(* Logix 5000 project; controller reports 1756-L63 rev 20.11; software revision 20.04; part 9 of 52 *)

        [41].log_data[16].valid := 1, [41].log_data[17].valid := 1, [41].log_data[18].valid := 1, [41].log_data[19].valid := 1, [41].time.Year := 2023, [41].time.Month := 1, [41].time.Day := 18, [41].time.Hour := 3, [41].time.Minute := 49, [41].time.Second := 59, [42].log_data[0].min := 1.0, [42].log_data[0].max := 1.0, [42].log_data[0].total := 300.0, [42].log_data[0].time := 300.0, [42].log_data[0].minminute := 50, [42].log_data[0].maxminute := 50, [42].log_data[0].valid := 1, [42].log_data[1].valid := 1, [42].log_data[2].valid := 1, [42].log_data[3].valid := 1, [42].log_data[4].valid := 1, [42].log_data[5].valid := 1, [42].log_data[6].valid := 1, [42].log_data[7].valid := 1, [42].log_data[8].valid := 1, [42].log_data[9].valid := 1, [42].log_data[10].valid := 1, [42].log_data[11].valid := 1, [42].log_data[12].valid := 1, [42].log_data[13].valid := 1, [42].log_data[14].valid := 1, [42].log_data[15].valid := 1, [42].log_data[16].valid := 1, [42].log_data[17].valid := 1, [42].log_data[18].valid := 1, [42].log_data[19].valid := 1, [42].time.Year := 2023, [42].time.Month := 1, [42].time.Day := 18, [42].time.Hour := 3, [42].time.Minute := 54, [42].time.Second := 59, [43].log_data[0].min := 1.0, [43].log_data[0].max := 1.0, [43].log_data[0].total := 300.0, [43].log_data[0].time := 300.0, [43].log_data[0].minminute := 55, [43].log_data[0].maxminute := 55, [43].log_data[0].valid := 1, [43].log_data[1].valid := 1, [43].log_data[2].valid := 1, [43].log_data[3].valid := 1, [43].log_data[4].valid := 1, [43].log_data[5].valid := 1, [43].log_data[6].valid := 1, [43].log_data[7].valid := 1, [43].log_data[8].valid := 1, [43].log_data[9].valid := 1, [43].log_data[10].valid := 1, [43].log_data[11].valid := 1,
        [43].log_data[12].valid := 1, [43].log_data[13].valid := 1, [43].log_data[14].valid := 1, [43].log_data[15].valid := 1, [43].log_data[16].valid := 1, [43].log_data[17].valid := 1, [43].log_data[18].valid := 1, [43].log_data[19].valid := 1, [43].time.Year := 2023, [43].time.Month := 1, [43].time.Day := 18, [43].time.Hour := 3, [43].time.Minute := 59, [43].time.Second := 59, [44].log_data[0].min := 1.0, [44].log_data[0].max := 1.0, [44].log_data[0].total := 300.0, [44].log_data[0].time := 300.0, [44].log_data[0].valid := 1, [44].log_data[1].valid := 1, [44].log_data[2].valid := 1, [44].log_data[3].valid := 1, [44].log_data[4].valid := 1, [44].log_data[5].valid := 1, [44].log_data[6].valid := 1, [44].log_data[7].valid := 1, [44].log_data[8].valid := 1, [44].log_data[9].valid := 1, [44].log_data[10].valid := 1, [44].log_data[11].valid := 1, [44].log_data[12].valid := 1, [44].log_data[13].valid := 1, [44].log_data[14].valid := 1, [44].log_data[15].valid := 1, [44].log_data[16].valid := 1, [44].log_data[17].valid := 1, [44].log_data[18].valid := 1, [44].log_data[19].valid := 1, [44].time.Year := 2023, [44].time.Month := 1, [44].time.Day := 18, [44].time.Hour := 4, [44].time.Minute := 4, [44].time.Second := 59, [45].log_data[0].min := 1.0, [45].log_data[0].max := 1.0, [45].log_data[0].total := 300.0, [45].log_data[0].time := 300.0, [45].log_data[0].minminute := 5, [45].log_data[0].maxminute := 5, [45].log_data[0].valid := 1, [45].log_data[1].valid := 1, [45].log_data[2].valid := 1, [45].log_data[3].valid := 1, [45].log_data[4].valid := 1, [45].log_data[5].valid := 1, [45].log_data[6].valid := 1, [45].log_data[7].valid := 1, [45].log_data[8].valid := 1, [45].log_data[9].valid := 1,
        [45].log_data[10].valid := 1, [45].log_data[11].valid := 1, [45].log_data[12].valid := 1, [45].log_data[13].valid := 1, [45].log_data[14].valid := 1, [45].log_data[15].valid := 1, [45].log_data[16].valid := 1, [45].log_data[17].valid := 1, [45].log_data[18].valid := 1, [45].log_data[19].valid := 1, [45].time.Year := 2023, [45].time.Month := 1, [45].time.Day := 18, [45].time.Hour := 4, [45].time.Minute := 9, [45].time.Second := 59, [46].log_data[0].min := 1.0, [46].log_data[0].max := 1.0, [46].log_data[0].total := 300.0, [46].log_data[0].time := 300.0, [46].log_data[0].minminute := 10, [46].log_data[0].maxminute := 10, [46].log_data[0].valid := 1, [46].log_data[1].valid := 1, [46].log_data[2].valid := 1, [46].log_data[3].valid := 1, [46].log_data[4].valid := 1, [46].log_data[5].valid := 1, [46].log_data[6].valid := 1, [46].log_data[7].valid := 1, [46].log_data[8].valid := 1, [46].log_data[9].valid := 1, [46].log_data[10].valid := 1, [46].log_data[11].valid := 1, [46].log_data[12].valid := 1, [46].log_data[13].valid := 1, [46].log_data[14].valid := 1, [46].log_data[15].valid := 1, [46].log_data[16].valid := 1, [46].log_data[17].valid := 1, [46].log_data[18].valid := 1, [46].log_data[19].valid := 1, [46].time.Year := 2023, [46].time.Month := 1, [46].time.Day := 18, [46].time.Hour := 4, [46].time.Minute := 14, [46].time.Second := 59, [47].log_data[0].min := 1.0, [47].log_data[0].max := 1.0, [47].log_data[0].total := 300.0, [47].log_data[0].time := 300.0, [47].log_data[0].minminute := 15, [47].log_data[0].maxminute := 15, [47].log_data[0].valid := 1, [47].log_data[1].valid := 1, [47].log_data[2].valid := 1, [47].log_data[3].valid := 1, [47].log_data[4].valid := 1, [47].log_data[5].valid := 1,
        [47].log_data[6].valid := 1, [47].log_data[7].valid := 1, [47].log_data[8].valid := 1, [47].log_data[9].valid := 1, [47].log_data[10].valid := 1, [47].log_data[11].valid := 1, [47].log_data[12].valid := 1, [47].log_data[13].valid := 1, [47].log_data[14].valid := 1, [47].log_data[15].valid := 1, [47].log_data[16].valid := 1, [47].log_data[17].valid := 1, [47].log_data[18].valid := 1, [47].log_data[19].valid := 1, [47].time.Year := 2023, [47].time.Month := 1, [47].time.Day := 18, [47].time.Hour := 4, [47].time.Minute := 19, [47].time.Second := 59, [48].log_data[0].min := 1.0, [48].log_data[0].max := 1.0, [48].log_data[0].total := 300.0, [48].log_data[0].time := 300.0, [48].log_data[0].minminute := 20, [48].log_data[0].maxminute := 20, [48].log_data[0].valid := 1, [48].log_data[1].valid := 1, [48].log_data[2].valid := 1, [48].log_data[3].valid := 1, [48].log_data[4].valid := 1, [48].log_data[5].valid := 1, [48].log_data[6].valid := 1, [48].log_data[7].valid := 1, [48].log_data[8].valid := 1, [48].log_data[9].valid := 1, [48].log_data[10].valid := 1, [48].log_data[11].valid := 1, [48].log_data[12].valid := 1, [48].log_data[13].valid := 1, [48].log_data[14].valid := 1, [48].log_data[15].valid := 1, [48].log_data[16].valid := 1, [48].log_data[17].valid := 1, [48].log_data[18].valid := 1, [48].log_data[19].valid := 1, [48].time.Year := 2023, [48].time.Month := 1, [48].time.Day := 18, [48].time.Hour := 4, [48].time.Minute := 24, [48].time.Second := 59, [49].log_data[0].min := 1.0, [49].log_data[0].max := 1.0, [49].log_data[0].total := 300.0, [49].log_data[0].time := 300.0, [49].log_data[0].minminute := 25, [49].log_data[0].maxminute := 25, [49].log_data[0].valid := 1, [49].log_data[1].valid := 1,
        [49].log_data[2].valid := 1, [49].log_data[3].valid := 1, [49].log_data[4].valid := 1, [49].log_data[5].valid := 1, [49].log_data[6].valid := 1, [49].log_data[7].valid := 1, [49].log_data[8].valid := 1, [49].log_data[9].valid := 1, [49].log_data[10].valid := 1, [49].log_data[11].valid := 1, [49].log_data[12].valid := 1, [49].log_data[13].valid := 1, [49].log_data[14].valid := 1, [49].log_data[15].valid := 1, [49].log_data[16].valid := 1, [49].log_data[17].valid := 1, [49].log_data[18].valid := 1, [49].log_data[19].valid := 1, [49].time.Year := 2023, [49].time.Month := 1, [49].time.Day := 18, [49].time.Hour := 4, [49].time.Minute := 29, [49].time.Second := 59, [50].log_data[0].min := 1.0, [50].log_data[0].max := 1.0, [50].log_data[0].total := 300.0, [50].log_data[0].time := 300.0, [50].log_data[0].minminute := 30, [50].log_data[0].maxminute := 30, [50].log_data[0].valid := 1, [50].log_data[1].valid := 1, [50].log_data[2].valid := 1, [50].log_data[3].valid := 1, [50].log_data[4].valid := 1, [50].log_data[5].valid := 1, [50].log_data[6].valid := 1, [50].log_data[7].valid := 1, [50].log_data[8].valid := 1, [50].log_data[9].valid := 1, [50].log_data[10].valid := 1, [50].log_data[11].valid := 1, [50].log_data[12].valid := 1, [50].log_data[13].valid := 1, [50].log_data[14].valid := 1, [50].log_data[15].valid := 1, [50].log_data[16].valid := 1, [50].log_data[17].valid := 1, [50].log_data[18].valid := 1, [50].log_data[19].valid := 1, [50].time.Year := 2023, [50].time.Month := 1, [50].time.Day := 18, [50].time.Hour := 4, [50].time.Minute := 34, [50].time.Second := 59, [51].log_data[0].min := 1.0, [51].log_data[0].max := 1.0, [51].log_data[0].total := 300.0, [51].log_data[0].time := 300.0,
        [51].log_data[0].minminute := 35, [51].log_data[0].maxminute := 35, [51].log_data[0].valid := 1, [51].log_data[1].valid := 1, [51].log_data[2].valid := 1, [51].log_data[3].valid := 1, [51].log_data[4].valid := 1, [51].log_data[5].valid := 1, [51].log_data[6].valid := 1, [51].log_data[7].valid := 1, [51].log_data[8].valid := 1, [51].log_data[9].valid := 1, [51].log_data[10].valid := 1, [51].log_data[11].valid := 1, [51].log_data[12].valid := 1, [51].log_data[13].valid := 1, [51].log_data[14].valid := 1, [51].log_data[15].valid := 1, [51].log_data[16].valid := 1, [51].log_data[17].valid := 1, [51].log_data[18].valid := 1, [51].log_data[19].valid := 1, [51].time.Year := 2023, [51].time.Month := 1, [51].time.Day := 18, [51].time.Hour := 4, [51].time.Minute := 39, [51].time.Second := 59, [52].log_data[0].min := 1.0, [52].log_data[0].max := 1.0, [52].log_data[0].total := 300.0, [52].log_data[0].time := 300.0, [52].log_data[0].minminute := 40, [52].log_data[0].maxminute := 40, [52].log_data[0].valid := 1, [52].log_data[1].valid := 1, [52].log_data[2].valid := 1, [52].log_data[3].valid := 1, [52].log_data[4].valid := 1, [52].log_data[5].valid := 1, [52].log_data[6].valid := 1, [52].log_data[7].valid := 1, [52].log_data[8].valid := 1, [52].log_data[9].valid := 1, [52].log_data[10].valid := 1, [52].log_data[11].valid := 1, [52].log_data[12].valid := 1, [52].log_data[13].valid := 1, [52].log_data[14].valid := 1, [52].log_data[15].valid := 1, [52].log_data[16].valid := 1, [52].log_data[17].valid := 1, [52].log_data[18].valid := 1, [52].log_data[19].valid := 1, [52].time.Year := 2023, [52].time.Month := 1, [52].time.Day := 18, [52].time.Hour := 4, [52].time.Minute := 44, [52].time.Second := 59,
        [53].log_data[0].min := 1.0, [53].log_data[0].max := 1.0, [53].log_data[0].total := 300.0, [53].log_data[0].time := 300.0, [53].log_data[0].minminute := 45, [53].log_data[0].maxminute := 45, [53].log_data[0].valid := 1, [53].log_data[1].valid := 1, [53].log_data[2].valid := 1, [53].log_data[3].valid := 1, [53].log_data[4].valid := 1, [53].log_data[5].valid := 1, [53].log_data[6].valid := 1, [53].log_data[7].valid := 1, [53].log_data[8].valid := 1, [53].log_data[9].valid := 1, [53].log_data[10].valid := 1, [53].log_data[11].valid := 1, [53].log_data[12].valid := 1, [53].log_data[13].valid := 1, [53].log_data[14].valid := 1, [53].log_data[15].valid := 1, [53].log_data[16].valid := 1, [53].log_data[17].valid := 1, [53].log_data[18].valid := 1, [53].log_data[19].valid := 1, [53].time.Year := 2023, [53].time.Month := 1, [53].time.Day := 18, [53].time.Hour := 4, [53].time.Minute := 49, [53].time.Second := 59, [54].log_data[0].min := 1.0, [54].log_data[0].max := 1.0, [54].log_data[0].total := 300.0, [54].log_data[0].time := 300.0, [54].log_data[0].minminute := 50, [54].log_data[0].maxminute := 50, [54].log_data[0].valid := 1, [54].log_data[1].valid := 1, [54].log_data[2].valid := 1, [54].log_data[3].valid := 1, [54].log_data[4].valid := 1, [54].log_data[5].valid := 1, [54].log_data[6].valid := 1, [54].log_data[7].valid := 1, [54].log_data[8].valid := 1, [54].log_data[9].valid := 1, [54].log_data[10].valid := 1, [54].log_data[11].valid := 1, [54].log_data[12].valid := 1, [54].log_data[13].valid := 1, [54].log_data[14].valid := 1, [54].log_data[15].valid := 1, [54].log_data[16].valid := 1, [54].log_data[17].valid := 1, [54].log_data[18].valid := 1, [54].log_data[19].valid := 1, [54].time.Year := 2023, [54].time.Month := 1,
        [54].time.Day := 18, [54].time.Hour := 4, [54].time.Minute := 54, [54].time.Second := 59, [55].log_data[0].min := 1.0, [55].log_data[0].max := 1.0, [55].log_data[0].total := 300.0, [55].log_data[0].time := 300.0, [55].log_data[0].minminute := 55, [55].log_data[0].maxminute := 55, [55].log_data[0].valid := 1, [55].log_data[1].valid := 1, [55].log_data[2].valid := 1, [55].log_data[3].valid := 1, [55].log_data[4].valid := 1, [55].log_data[5].valid := 1, [55].log_data[6].valid := 1, [55].log_data[7].valid := 1, [55].log_data[8].valid := 1, [55].log_data[9].valid := 1, [55].log_data[10].valid := 1, [55].log_data[11].valid := 1, [55].log_data[12].valid := 1, [55].log_data[13].valid := 1, [55].log_data[14].valid := 1, [55].log_data[15].valid := 1, [55].log_data[16].valid := 1, [55].log_data[17].valid := 1, [55].log_data[18].valid := 1, [55].log_data[19].valid := 1, [55].time.Year := 2023, [55].time.Month := 1, [55].time.Day := 18, [55].time.Hour := 4, [55].time.Minute := 59, [55].time.Second := 59, [56].log_data[0].min := 1.0, [56].log_data[0].max := 1.0, [56].log_data[0].total := 300.0, [56].log_data[0].time := 300.0, [56].log_data[0].valid := 1, [56].log_data[1].valid := 1, [56].log_data[2].valid := 1, [56].log_data[3].valid := 1, [56].log_data[4].valid := 1, [56].log_data[5].valid := 1, [56].log_data[6].valid := 1, [56].log_data[7].valid := 1, [56].log_data[8].valid := 1, [56].log_data[9].valid := 1, [56].log_data[10].valid := 1, [56].log_data[11].valid := 1, [56].log_data[12].valid := 1, [56].log_data[13].valid := 1, [56].log_data[14].valid := 1, [56].log_data[15].valid := 1, [56].log_data[16].valid := 1, [56].log_data[17].valid := 1, [56].log_data[18].valid := 1, [56].log_data[19].valid := 1,
        [56].time.Year := 2023, [56].time.Month := 1, [56].time.Day := 18, [56].time.Hour := 5, [56].time.Minute := 4, [56].time.Second := 59, [57].log_data[0].min := 1.0, [57].log_data[0].max := 1.0, [57].log_data[0].total := 300.0, [57].log_data[0].time := 300.0, [57].log_data[0].minminute := 5, [57].log_data[0].maxminute := 5, [57].log_data[0].valid := 1, [57].log_data[1].valid := 1, [57].log_data[2].valid := 1, [57].log_data[3].valid := 1, [57].log_data[4].valid := 1, [57].log_data[5].valid := 1, [57].log_data[6].valid := 1, [57].log_data[7].valid := 1, [57].log_data[8].valid := 1, [57].log_data[9].valid := 1, [57].log_data[10].valid := 1, [57].log_data[11].valid := 1, [57].log_data[12].valid := 1, [57].log_data[13].valid := 1, [57].log_data[14].valid := 1, [57].log_data[15].valid := 1, [57].log_data[16].valid := 1, [57].log_data[17].valid := 1, [57].log_data[18].valid := 1, [57].log_data[19].valid := 1, [57].time.Year := 2023, [57].time.Month := 1, [57].time.Day := 18, [57].time.Hour := 5, [57].time.Minute := 9, [57].time.Second := 59, [58].log_data[0].min := 1.0, [58].log_data[0].max := 1.0, [58].log_data[0].total := 300.0, [58].log_data[0].time := 300.0, [58].log_data[0].minminute := 10, [58].log_data[0].maxminute := 10, [58].log_data[0].valid := 1, [58].log_data[1].valid := 1, [58].log_data[2].valid := 1, [58].log_data[3].valid := 1, [58].log_data[4].valid := 1, [58].log_data[5].valid := 1, [58].log_data[6].valid := 1, [58].log_data[7].valid := 1, [58].log_data[8].valid := 1, [58].log_data[9].valid := 1, [58].log_data[10].valid := 1, [58].log_data[11].valid := 1, [58].log_data[12].valid := 1, [58].log_data[13].valid := 1, [58].log_data[14].valid := 1, [58].log_data[15].valid := 1,
        [58].log_data[16].valid := 1, [58].log_data[17].valid := 1, [58].log_data[18].valid := 1, [58].log_data[19].valid := 1, [58].time.Year := 2023, [58].time.Month := 1, [58].time.Day := 18, [58].time.Hour := 5, [58].time.Minute := 14, [58].time.Second := 59, [59].log_data[0].min := 1.0, [59].log_data[0].max := 1.0, [59].log_data[0].total := 300.0, [59].log_data[0].time := 300.0, [59].log_data[0].minminute := 15, [59].log_data[0].maxminute := 15, [59].log_data[0].valid := 1, [59].log_data[1].valid := 1, [59].log_data[2].valid := 1, [59].log_data[3].valid := 1, [59].log_data[4].valid := 1, [59].log_data[5].valid := 1, [59].log_data[6].valid := 1, [59].log_data[7].valid := 1, [59].log_data[8].valid := 1, [59].log_data[9].valid := 1, [59].log_data[10].valid := 1, [59].log_data[11].valid := 1, [59].log_data[12].valid := 1, [59].log_data[13].valid := 1, [59].log_data[14].valid := 1, [59].log_data[15].valid := 1, [59].log_data[16].valid := 1, [59].log_data[17].valid := 1, [59].log_data[18].valid := 1, [59].log_data[19].valid := 1, [59].time.Year := 2023, [59].time.Month := 1, [59].time.Day := 18, [59].time.Hour := 5, [59].time.Minute := 19, [59].time.Second := 59, [60].log_data[0].min := 1.0, [60].log_data[0].max := 1.0, [60].log_data[0].total := 300.0, [60].log_data[0].time := 300.0, [60].log_data[0].minminute := 20, [60].log_data[0].maxminute := 20, [60].log_data[0].valid := 1, [60].log_data[1].valid := 1, [60].log_data[2].valid := 1, [60].log_data[3].valid := 1, [60].log_data[4].valid := 1, [60].log_data[5].valid := 1, [60].log_data[6].valid := 1, [60].log_data[7].valid := 1, [60].log_data[8].valid := 1, [60].log_data[9].valid := 1, [60].log_data[10].valid := 1, [60].log_data[11].valid := 1,
        [60].log_data[12].valid := 1, [60].log_data[13].valid := 1, [60].log_data[14].valid := 1, [60].log_data[15].valid := 1, [60].log_data[16].valid := 1, [60].log_data[17].valid := 1, [60].log_data[18].valid := 1, [60].log_data[19].valid := 1, [60].time.Year := 2023, [60].time.Month := 1, [60].time.Day := 18, [60].time.Hour := 5, [60].time.Minute := 24, [60].time.Second := 59, [61].log_data[0].min := 1.0, [61].log_data[0].max := 1.0, [61].log_data[0].total := 300.0, [61].log_data[0].time := 300.0, [61].log_data[0].minminute := 25, [61].log_data[0].maxminute := 25, [61].log_data[0].valid := 1, [61].log_data[1].valid := 1, [61].log_data[2].valid := 1, [61].log_data[3].valid := 1, [61].log_data[4].valid := 1, [61].log_data[5].valid := 1, [61].log_data[6].valid := 1, [61].log_data[7].valid := 1, [61].log_data[8].valid := 1, [61].log_data[9].valid := 1, [61].log_data[10].valid := 1, [61].log_data[11].valid := 1, [61].log_data[12].valid := 1, [61].log_data[13].valid := 1, [61].log_data[14].valid := 1, [61].log_data[15].valid := 1, [61].log_data[16].valid := 1, [61].log_data[17].valid := 1, [61].log_data[18].valid := 1, [61].log_data[19].valid := 1, [61].time.Year := 2023, [61].time.Month := 1, [61].time.Day := 18, [61].time.Hour := 5, [61].time.Minute := 29, [61].time.Second := 59, [62].log_data[0].min := 1.0, [62].log_data[0].max := 1.0, [62].log_data[0].total := 300.0, [62].log_data[0].time := 300.0, [62].log_data[0].minminute := 30, [62].log_data[0].maxminute := 30, [62].log_data[0].valid := 1, [62].log_data[1].valid := 1, [62].log_data[2].valid := 1, [62].log_data[3].valid := 1, [62].log_data[4].valid := 1, [62].log_data[5].valid := 1, [62].log_data[6].valid := 1, [62].log_data[7].valid := 1,
        [62].log_data[8].valid := 1, [62].log_data[9].valid := 1, [62].log_data[10].valid := 1, [62].log_data[11].valid := 1, [62].log_data[12].valid := 1, [62].log_data[13].valid := 1, [62].log_data[14].valid := 1, [62].log_data[15].valid := 1, [62].log_data[16].valid := 1, [62].log_data[17].valid := 1, [62].log_data[18].valid := 1, [62].log_data[19].valid := 1, [62].time.Year := 2023, [62].time.Month := 1, [62].time.Day := 18, [62].time.Hour := 5, [62].time.Minute := 34, [62].time.Second := 59, [63].log_data[0].min := 1.0, [63].log_data[0].max := 1.0, [63].log_data[0].total := 300.0, [63].log_data[0].time := 300.0, [63].log_data[0].minminute := 35, [63].log_data[0].maxminute := 35, [63].log_data[0].valid := 1, [63].log_data[1].valid := 1, [63].log_data[2].valid := 1, [63].log_data[3].valid := 1, [63].log_data[4].valid := 1, [63].log_data[5].valid := 1, [63].log_data[6].valid := 1, [63].log_data[7].valid := 1, [63].log_data[8].valid := 1, [63].log_data[9].valid := 1, [63].log_data[10].valid := 1, [63].log_data[11].valid := 1, [63].log_data[12].valid := 1, [63].log_data[13].valid := 1, [63].log_data[14].valid := 1, [63].log_data[15].valid := 1, [63].log_data[16].valid := 1, [63].log_data[17].valid := 1, [63].log_data[18].valid := 1, [63].log_data[19].valid := 1, [63].time.Year := 2023, [63].time.Month := 1, [63].time.Day := 18, [63].time.Hour := 5, [63].time.Minute := 39, [63].time.Second := 59, [64].log_data[0].min := 1.0, [64].log_data[0].max := 1.0, [64].log_data[0].total := 300.0, [64].log_data[0].time := 300.0, [64].log_data[0].minminute := 40, [64].log_data[0].maxminute := 40, [64].log_data[0].valid := 1, [64].log_data[1].valid := 1, [64].log_data[2].valid := 1, [64].log_data[3].valid := 1,
        [64].log_data[4].valid := 1, [64].log_data[5].valid := 1, [64].log_data[6].valid := 1, [64].log_data[7].valid := 1, [64].log_data[8].valid := 1, [64].log_data[9].valid := 1, [64].log_data[10].valid := 1, [64].log_data[11].valid := 1, [64].log_data[12].valid := 1, [64].log_data[13].valid := 1, [64].log_data[14].valid := 1, [64].log_data[15].valid := 1, [64].log_data[16].valid := 1, [64].log_data[17].valid := 1, [64].log_data[18].valid := 1, [64].log_data[19].valid := 1, [64].time.Year := 2023, [64].time.Month := 1, [64].time.Day := 18, [64].time.Hour := 5, [64].time.Minute := 44, [64].time.Second := 59, [65].log_data[0].min := 1.0, [65].log_data[0].max := 1.0, [65].log_data[0].total := 300.0, [65].log_data[0].time := 300.0, [65].log_data[0].minminute := 45, [65].log_data[0].maxminute := 45, [65].log_data[0].valid := 1, [65].log_data[1].valid := 1, [65].log_data[2].valid := 1, [65].log_data[3].valid := 1, [65].log_data[4].valid := 1, [65].log_data[5].valid := 1, [65].log_data[6].valid := 1, [65].log_data[7].valid := 1, [65].log_data[8].valid := 1, [65].log_data[9].valid := 1, [65].log_data[10].valid := 1, [65].log_data[11].valid := 1, [65].log_data[12].valid := 1, [65].log_data[13].valid := 1, [65].log_data[14].valid := 1, [65].log_data[15].valid := 1, [65].log_data[16].valid := 1, [65].log_data[17].valid := 1, [65].log_data[18].valid := 1, [65].log_data[19].valid := 1, [65].time.Year := 2023, [65].time.Month := 1, [65].time.Day := 18, [65].time.Hour := 5, [65].time.Minute := 49, [65].time.Second := 59, [66].log_data[0].min := 1.0, [66].log_data[0].max := 1.0, [66].log_data[0].total := 300.0, [66].log_data[0].time := 300.0, [66].log_data[0].minminute := 50, [66].log_data[0].maxminute := 50,
        [66].log_data[0].valid := 1, [66].log_data[1].valid := 1, [66].log_data[2].valid := 1, [66].log_data[3].valid := 1, [66].log_data[4].valid := 1, [66].log_data[5].valid := 1, [66].log_data[6].valid := 1, [66].log_data[7].valid := 1, [66].log_data[8].valid := 1, [66].log_data[9].valid := 1, [66].log_data[10].valid := 1, [66].log_data[11].valid := 1, [66].log_data[12].valid := 1, [66].log_data[13].valid := 1, [66].log_data[14].valid := 1, [66].log_data[15].valid := 1, [66].log_data[16].valid := 1, [66].log_data[17].valid := 1, [66].log_data[18].valid := 1, [66].log_data[19].valid := 1, [66].time.Year := 2023, [66].time.Month := 1, [66].time.Day := 18, [66].time.Hour := 5, [66].time.Minute := 54, [66].time.Second := 59, [67].log_data[0].min := 1.0, [67].log_data[0].max := 1.0, [67].log_data[0].total := 300.0, [67].log_data[0].time := 300.0, [67].log_data[0].minminute := 55, [67].log_data[0].maxminute := 55, [67].log_data[0].valid := 1, [67].log_data[1].valid := 1, [67].log_data[2].valid := 1, [67].log_data[3].valid := 1, [67].log_data[4].valid := 1, [67].log_data[5].valid := 1, [67].log_data[6].valid := 1, [67].log_data[7].valid := 1, [67].log_data[8].valid := 1, [67].log_data[9].valid := 1, [67].log_data[10].valid := 1, [67].log_data[11].valid := 1, [67].log_data[12].valid := 1, [67].log_data[13].valid := 1, [67].log_data[14].valid := 1, [67].log_data[15].valid := 1, [67].log_data[16].valid := 1, [67].log_data[17].valid := 1, [67].log_data[18].valid := 1, [67].log_data[19].valid := 1, [67].time.Year := 2023, [67].time.Month := 1, [67].time.Day := 18, [67].time.Hour := 5, [67].time.Minute := 59, [67].time.Second := 59, [68].log_data[0].min := 1.0, [68].log_data[0].max := 1.0,
        [68].log_data[0].total := 300.0, [68].log_data[0].time := 300.0, [68].log_data[0].valid := 1, [68].log_data[1].valid := 1, [68].log_data[2].valid := 1, [68].log_data[3].valid := 1, [68].log_data[4].valid := 1, [68].log_data[5].valid := 1, [68].log_data[6].valid := 1, [68].log_data[7].valid := 1, [68].log_data[8].valid := 1, [68].log_data[9].valid := 1, [68].log_data[10].valid := 1, [68].log_data[11].valid := 1, [68].log_data[12].valid := 1, [68].log_data[13].valid := 1, [68].log_data[14].valid := 1, [68].log_data[15].valid := 1, [68].log_data[16].valid := 1, [68].log_data[17].valid := 1, [68].log_data[18].valid := 1, [68].log_data[19].valid := 1, [68].time.Year := 2023, [68].time.Month := 1, [68].time.Day := 18, [68].time.Hour := 6, [68].time.Minute := 4, [68].time.Second := 59, [69].log_data[0].min := 1.0, [69].log_data[0].max := 1.0, [69].log_data[0].total := 300.0, [69].log_data[0].time := 300.0, [69].log_data[0].minminute := 5, [69].log_data[0].maxminute := 5, [69].log_data[0].valid := 1, [69].log_data[1].valid := 1, [69].log_data[2].valid := 1, [69].log_data[3].valid := 1, [69].log_data[4].valid := 1, [69].log_data[5].valid := 1, [69].log_data[6].valid := 1, [69].log_data[7].valid := 1, [69].log_data[8].valid := 1, [69].log_data[9].valid := 1, [69].log_data[10].valid := 1, [69].log_data[11].valid := 1, [69].log_data[12].valid := 1, [69].log_data[13].valid := 1, [69].log_data[14].valid := 1, [69].log_data[15].valid := 1, [69].log_data[16].valid := 1, [69].log_data[17].valid := 1, [69].log_data[18].valid := 1, [69].log_data[19].valid := 1, [69].time.Year := 2023, [69].time.Month := 1, [69].time.Day := 18, [69].time.Hour := 6, [69].time.Minute := 9, [69].time.Second := 59,
        [70].log_data[0].min := 1.0, [70].log_data[0].max := 1.0, [70].log_data[0].total := 300.0, [70].log_data[0].time := 300.0, [70].log_data[0].minminute := 10, [70].log_data[0].maxminute := 10, [70].log_data[0].valid := 1, [70].log_data[1].valid := 1, [70].log_data[2].valid := 1, [70].log_data[3].valid := 1, [70].log_data[4].valid := 1, [70].log_data[5].valid := 1, [70].log_data[6].valid := 1, [70].log_data[7].valid := 1, [70].log_data[8].valid := 1, [70].log_data[9].valid := 1, [70].log_data[10].valid := 1, [70].log_data[11].valid := 1, [70].log_data[12].valid := 1, [70].log_data[13].valid := 1, [70].log_data[14].valid := 1, [70].log_data[15].valid := 1, [70].log_data[16].valid := 1, [70].log_data[17].valid := 1, [70].log_data[18].valid := 1, [70].log_data[19].valid := 1, [70].time.Year := 2023, [70].time.Month := 1, [70].time.Day := 18, [70].time.Hour := 6, [70].time.Minute := 14, [70].time.Second := 59, [71].log_data[0].min := 1.0, [71].log_data[0].max := 1.0, [71].log_data[0].total := 300.0, [71].log_data[0].time := 300.0, [71].log_data[0].minminute := 15, [71].log_data[0].maxminute := 15, [71].log_data[0].valid := 1, [71].log_data[1].valid := 1, [71].log_data[2].valid := 1, [71].log_data[3].valid := 1, [71].log_data[4].valid := 1, [71].log_data[5].valid := 1, [71].log_data[6].valid := 1, [71].log_data[7].valid := 1, [71].log_data[8].valid := 1, [71].log_data[9].valid := 1, [71].log_data[10].valid := 1, [71].log_data[11].valid := 1, [71].log_data[12].valid := 1, [71].log_data[13].valid := 1, [71].log_data[14].valid := 1, [71].log_data[15].valid := 1, [71].log_data[16].valid := 1, [71].log_data[17].valid := 1, [71].log_data[18].valid := 1, [71].log_data[19].valid := 1, [71].time.Year := 2023, [71].time.Month := 1,
        [71].time.Day := 18, [71].time.Hour := 6, [71].time.Minute := 19, [71].time.Second := 59, [72].log_data[0].min := 1.0, [72].log_data[0].max := 1.0, [72].log_data[0].total := 300.0, [72].log_data[0].time := 300.0, [72].log_data[0].minminute := 20, [72].log_data[0].maxminute := 20, [72].log_data[0].valid := 1, [72].log_data[1].valid := 1, [72].log_data[2].valid := 1, [72].log_data[3].valid := 1, [72].log_data[4].valid := 1, [72].log_data[5].valid := 1, [72].log_data[6].valid := 1, [72].log_data[7].valid := 1, [72].log_data[8].valid := 1, [72].log_data[9].valid := 1, [72].log_data[10].valid := 1, [72].log_data[11].valid := 1, [72].log_data[12].valid := 1, [72].log_data[13].valid := 1, [72].log_data[14].valid := 1, [72].log_data[15].valid := 1, [72].log_data[16].valid := 1, [72].log_data[17].valid := 1, [72].log_data[18].valid := 1, [72].log_data[19].valid := 1, [72].time.Year := 2023, [72].time.Month := 1, [72].time.Day := 18, [72].time.Hour := 6, [72].time.Minute := 24, [72].time.Second := 59, [73].log_data[0].min := 1.0, [73].log_data[0].max := 1.0, [73].log_data[0].total := 300.0, [73].log_data[0].time := 300.0, [73].log_data[0].minminute := 25, [73].log_data[0].maxminute := 25, [73].log_data[0].valid := 1, [73].log_data[1].valid := 1, [73].log_data[2].valid := 1, [73].log_data[3].valid := 1, [73].log_data[4].valid := 1, [73].log_data[5].valid := 1, [73].log_data[6].valid := 1, [73].log_data[7].valid := 1, [73].log_data[8].valid := 1, [73].log_data[9].valid := 1, [73].log_data[10].valid := 1, [73].log_data[11].valid := 1, [73].log_data[12].valid := 1, [73].log_data[13].valid := 1, [73].log_data[14].valid := 1, [73].log_data[15].valid := 1, [73].log_data[16].valid := 1, [73].log_data[17].valid := 1,
        [73].log_data[18].valid := 1, [73].log_data[19].valid := 1, [73].time.Year := 2023, [73].time.Month := 1, [73].time.Day := 18, [73].time.Hour := 6, [73].time.Minute := 29, [73].time.Second := 59, [74].log_data[0].min := 1.0, [74].log_data[0].max := 1.0, [74].log_data[0].total := 300.0, [74].log_data[0].time := 300.0, [74].log_data[0].minminute := 30, [74].log_data[0].maxminute := 30, [74].log_data[0].valid := 1, [74].log_data[1].valid := 1, [74].log_data[2].valid := 1, [74].log_data[3].valid := 1, [74].log_data[4].valid := 1, [74].log_data[5].valid := 1, [74].log_data[6].valid := 1, [74].log_data[7].valid := 1, [74].log_data[8].valid := 1, [74].log_data[9].valid := 1, [74].log_data[10].valid := 1, [74].log_data[11].valid := 1, [74].log_data[12].valid := 1, [74].log_data[13].valid := 1, [74].log_data[14].valid := 1, [74].log_data[15].valid := 1, [74].log_data[16].valid := 1, [74].log_data[17].valid := 1, [74].log_data[18].valid := 1, [74].log_data[19].valid := 1, [74].time.Year := 2023, [74].time.Month := 1, [74].time.Day := 18, [74].time.Hour := 6, [74].time.Minute := 34, [74].time.Second := 59, [75].log_data[0].min := 1.0, [75].log_data[0].max := 1.0, [75].log_data[0].total := 300.0, [75].log_data[0].time := 300.0, [75].log_data[0].minminute := 35, [75].log_data[0].maxminute := 35, [75].log_data[0].valid := 1, [75].log_data[1].valid := 1, [75].log_data[2].valid := 1, [75].log_data[3].valid := 1, [75].log_data[4].valid := 1, [75].log_data[5].valid := 1, [75].log_data[6].valid := 1, [75].log_data[7].valid := 1, [75].log_data[8].valid := 1, [75].log_data[9].valid := 1, [75].log_data[10].valid := 1, [75].log_data[11].valid := 1, [75].log_data[12].valid := 1, [75].log_data[13].valid := 1,
        [75].log_data[14].valid := 1, [75].log_data[15].valid := 1, [75].log_data[16].valid := 1, [75].log_data[17].valid := 1, [75].log_data[18].valid := 1, [75].log_data[19].valid := 1, [75].time.Year := 2023, [75].time.Month := 1, [75].time.Day := 18, [75].time.Hour := 6, [75].time.Minute := 39, [75].time.Second := 59, [76].log_data[0].min := 1.0, [76].log_data[0].max := 1.0, [76].log_data[0].total := 300.0, [76].log_data[0].time := 300.0, [76].log_data[0].minminute := 40, [76].log_data[0].maxminute := 40, [76].log_data[0].valid := 1, [76].log_data[1].valid := 1, [76].log_data[2].valid := 1, [76].log_data[3].valid := 1, [76].log_data[4].valid := 1, [76].log_data[5].valid := 1, [76].log_data[6].valid := 1, [76].log_data[7].valid := 1, [76].log_data[8].valid := 1, [76].log_data[9].valid := 1, [76].log_data[10].valid := 1, [76].log_data[11].valid := 1, [76].log_data[12].valid := 1, [76].log_data[13].valid := 1, [76].log_data[14].valid := 1, [76].log_data[15].valid := 1, [76].log_data[16].valid := 1, [76].log_data[17].valid := 1, [76].log_data[18].valid := 1, [76].log_data[19].valid := 1, [76].time.Year := 2023, [76].time.Month := 1, [76].time.Day := 18, [76].time.Hour := 6, [76].time.Minute := 44, [76].time.Second := 59, [77].log_data[0].min := 1.0, [77].log_data[0].max := 1.0, [77].log_data[0].total := 300.0, [77].log_data[0].time := 300.0, [77].log_data[0].minminute := 45, [77].log_data[0].maxminute := 45, [77].log_data[0].valid := 1, [77].log_data[1].valid := 1, [77].log_data[2].valid := 1, [77].log_data[3].valid := 1, [77].log_data[4].valid := 1, [77].log_data[5].valid := 1, [77].log_data[6].valid := 1, [77].log_data[7].valid := 1, [77].log_data[8].valid := 1, [77].log_data[9].valid := 1,
        [77].log_data[10].valid := 1, [77].log_data[11].valid := 1, [77].log_data[12].valid := 1, [77].log_data[13].valid := 1, [77].log_data[14].valid := 1, [77].log_data[15].valid := 1, [77].log_data[16].valid := 1, [77].log_data[17].valid := 1, [77].log_data[18].valid := 1, [77].log_data[19].valid := 1, [77].time.Year := 2023, [77].time.Month := 1, [77].time.Day := 18, [77].time.Hour := 6, [77].time.Minute := 49, [77].time.Second := 59, [78].log_data[0].min := 1.0, [78].log_data[0].max := 1.0, [78].log_data[0].total := 300.0, [78].log_data[0].time := 300.0, [78].log_data[0].minminute := 50, [78].log_data[0].maxminute := 50, [78].log_data[0].valid := 1, [78].log_data[1].valid := 1, [78].log_data[2].valid := 1, [78].log_data[3].valid := 1, [78].log_data[4].valid := 1, [78].log_data[5].valid := 1, [78].log_data[6].valid := 1, [78].log_data[7].valid := 1, [78].log_data[8].valid := 1, [78].log_data[9].valid := 1, [78].log_data[10].valid := 1, [78].log_data[11].valid := 1, [78].log_data[12].valid := 1, [78].log_data[13].valid := 1, [78].log_data[14].valid := 1, [78].log_data[15].valid := 1, [78].log_data[16].valid := 1, [78].log_data[17].valid := 1, [78].log_data[18].valid := 1, [78].log_data[19].valid := 1, [78].time.Year := 2023, [78].time.Month := 1, [78].time.Day := 18, [78].time.Hour := 6, [78].time.Minute := 54, [78].time.Second := 59, [79].log_data[0].min := 1.0, [79].log_data[0].max := 1.0, [79].log_data[0].total := 300.0, [79].log_data[0].time := 300.0, [79].log_data[0].minminute := 55, [79].log_data[0].maxminute := 55, [79].log_data[0].valid := 1, [79].log_data[1].valid := 1, [79].log_data[2].valid := 1, [79].log_data[3].valid := 1, [79].log_data[4].valid := 1, [79].log_data[5].valid := 1,
        [79].log_data[6].valid := 1, [79].log_data[7].valid := 1, [79].log_data[8].valid := 1, [79].log_data[9].valid := 1, [79].log_data[10].valid := 1, [79].log_data[11].valid := 1, [79].log_data[12].valid := 1, [79].log_data[13].valid := 1, [79].log_data[14].valid := 1, [79].log_data[15].valid := 1, [79].log_data[16].valid := 1, [79].log_data[17].valid := 1, [79].log_data[18].valid := 1, [79].log_data[19].valid := 1, [79].time.Year := 2023, [79].time.Month := 1, [79].time.Day := 18, [79].time.Hour := 6, [79].time.Minute := 59, [79].time.Second := 59, [80].log_data[0].min := 1.0, [80].log_data[0].max := 1.0, [80].log_data[0].total := 300.0, [80].log_data[0].time := 300.0, [80].log_data[0].valid := 1, [80].log_data[1].valid := 1, [80].log_data[2].valid := 1, [80].log_data[3].valid := 1, [80].log_data[4].valid := 1, [80].log_data[5].valid := 1, [80].log_data[6].valid := 1, [80].log_data[7].valid := 1, [80].log_data[8].valid := 1, [80].log_data[9].valid := 1, [80].log_data[10].valid := 1, [80].log_data[11].valid := 1, [80].log_data[12].valid := 1, [80].log_data[13].valid := 1, [80].log_data[14].valid := 1, [80].log_data[15].valid := 1, [80].log_data[16].valid := 1, [80].log_data[17].valid := 1, [80].log_data[18].valid := 1, [80].log_data[19].valid := 1, [80].time.Year := 2023, [80].time.Month := 1, [80].time.Day := 18, [80].time.Hour := 7, [80].time.Minute := 4, [80].time.Second := 59, [81].log_data[0].min := 1.0, [81].log_data[0].max := 1.0, [81].log_data[0].total := 300.0, [81].log_data[0].time := 300.0, [81].log_data[0].minminute := 5, [81].log_data[0].maxminute := 5, [81].log_data[0].valid := 1, [81].log_data[1].valid := 1, [81].log_data[2].valid := 1, [81].log_data[3].valid := 1,
        [81].log_data[4].valid := 1, [81].log_data[5].valid := 1, [81].log_data[6].valid := 1, [81].log_data[7].valid := 1, [81].log_data[8].valid := 1, [81].log_data[9].valid := 1, [81].log_data[10].valid := 1, [81].log_data[11].valid := 1, [81].log_data[12].valid := 1, [81].log_data[13].valid := 1, [81].log_data[14].valid := 1, [81].log_data[15].valid := 1, [81].log_data[16].valid := 1, [81].log_data[17].valid := 1, [81].log_data[18].valid := 1, [81].log_data[19].valid := 1, [81].time.Year := 2023, [81].time.Month := 1, [81].time.Day := 18, [81].time.Hour := 7, [81].time.Minute := 9, [81].time.Second := 59, [82].log_data[0].min := 1.0, [82].log_data[0].max := 1.0, [82].log_data[0].total := 300.0, [82].log_data[0].time := 300.0, [82].log_data[0].minminute := 10, [82].log_data[0].maxminute := 10, [82].log_data[0].valid := 1, [82].log_data[1].valid := 1, [82].log_data[2].valid := 1, [82].log_data[3].valid := 1, [82].log_data[4].valid := 1, [82].log_data[5].valid := 1, [82].log_data[6].valid := 1, [82].log_data[7].valid := 1, [82].log_data[8].valid := 1, [82].log_data[9].valid := 1, [82].log_data[10].valid := 1, [82].log_data[11].valid := 1, [82].log_data[12].valid := 1, [82].log_data[13].valid := 1, [82].log_data[14].valid := 1, [82].log_data[15].valid := 1, [82].log_data[16].valid := 1, [82].log_data[17].valid := 1, [82].log_data[18].valid := 1, [82].log_data[19].valid := 1, [82].time.Year := 2023, [82].time.Month := 1, [82].time.Day := 18, [82].time.Hour := 7, [82].time.Minute := 14, [82].time.Second := 59, [83].log_data[0].min := 1.0, [83].log_data[0].max := 1.0, [83].log_data[0].total := 300.0, [83].log_data[0].time := 300.0, [83].log_data[0].minminute := 15, [83].log_data[0].maxminute := 15,
        [83].log_data[0].valid := 1, [83].log_data[1].valid := 1, [83].log_data[2].valid := 1, [83].log_data[3].valid := 1, [83].log_data[4].valid := 1, [83].log_data[5].valid := 1, [83].log_data[6].valid := 1, [83].log_data[7].valid := 1, [83].log_data[8].valid := 1, [83].log_data[9].valid := 1, [83].log_data[10].valid := 1, [83].log_data[11].valid := 1, [83].log_data[12].valid := 1, [83].log_data[13].valid := 1, [83].log_data[14].valid := 1, [83].log_data[15].valid := 1, [83].log_data[16].valid := 1, [83].log_data[17].valid := 1, [83].log_data[18].valid := 1, [83].log_data[19].valid := 1, [83].time.Year := 2023, [83].time.Month := 1, [83].time.Day := 18, [83].time.Hour := 7, [83].time.Minute := 19, [83].time.Second := 59, [84].log_data[0].min := 1.0, [84].log_data[0].max := 1.0, [84].log_data[0].total := 300.0, [84].log_data[0].time := 300.0, [84].log_data[0].minminute := 20, [84].log_data[0].maxminute := 20, [84].log_data[0].valid := 1, [84].log_data[1].valid := 1, [84].log_data[2].valid := 1, [84].log_data[3].valid := 1, [84].log_data[4].valid := 1, [84].log_data[5].valid := 1, [84].log_data[6].valid := 1, [84].log_data[7].valid := 1, [84].log_data[8].valid := 1, [84].log_data[9].valid := 1, [84].log_data[10].valid := 1, [84].log_data[11].valid := 1, [84].log_data[12].valid := 1, [84].log_data[13].valid := 1, [84].log_data[14].valid := 1, [84].log_data[15].valid := 1, [84].log_data[16].valid := 1, [84].log_data[17].valid := 1, [84].log_data[18].valid := 1, [84].log_data[19].valid := 1, [84].time.Year := 2023, [84].time.Month := 1, [84].time.Day := 18, [84].time.Hour := 7, [84].time.Minute := 24, [84].time.Second := 59, [85].log_data[0].min := 1.0, [85].log_data[0].max := 1.0,
        [85].log_data[0].total := 300.0, [85].log_data[0].time := 300.0, [85].log_data[0].minminute := 25, [85].log_data[0].maxminute := 25, [85].log_data[0].valid := 1, [85].log_data[1].valid := 1, [85].log_data[2].valid := 1, [85].log_data[3].valid := 1, [85].log_data[4].valid := 1, [85].log_data[5].valid := 1, [85].log_data[6].valid := 1, [85].log_data[7].valid := 1, [85].log_data[8].valid := 1, [85].log_data[9].valid := 1, [85].log_data[10].valid := 1, [85].log_data[11].valid := 1, [85].log_data[12].valid := 1, [85].log_data[13].valid := 1, [85].log_data[14].valid := 1, [85].log_data[15].valid := 1, [85].log_data[16].valid := 1, [85].log_data[17].valid := 1, [85].log_data[18].valid := 1, [85].log_data[19].valid := 1, [85].time.Year := 2023, [85].time.Month := 1, [85].time.Day := 18, [85].time.Hour := 7, [85].time.Minute := 29, [85].time.Second := 59, [86].log_data[0].min := 1.0, [86].log_data[0].max := 1.0, [86].log_data[0].total := 300.0, [86].log_data[0].time := 300.0, [86].log_data[0].minminute := 30, [86].log_data[0].maxminute := 30, [86].log_data[0].valid := 1, [86].log_data[1].valid := 1, [86].log_data[2].valid := 1, [86].log_data[3].valid := 1, [86].log_data[4].valid := 1, [86].log_data[5].valid := 1, [86].log_data[6].valid := 1, [86].log_data[7].valid := 1, [86].log_data[8].valid := 1, [86].log_data[9].valid := 1, [86].log_data[10].valid := 1, [86].log_data[11].valid := 1, [86].log_data[12].valid := 1, [86].log_data[13].valid := 1, [86].log_data[14].valid := 1, [86].log_data[15].valid := 1, [86].log_data[16].valid := 1, [86].log_data[17].valid := 1, [86].log_data[18].valid := 1, [86].log_data[19].valid := 1, [86].time.Year := 2023, [86].time.Month := 1, [86].time.Day := 18, [86].time.Hour := 7,
        [86].time.Minute := 34, [86].time.Second := 59, [87].log_data[0].min := 1.0, [87].log_data[0].max := 1.0, [87].log_data[0].total := 300.0, [87].log_data[0].time := 300.0, [87].log_data[0].minminute := 35, [87].log_data[0].maxminute := 35, [87].log_data[0].valid := 1, [87].log_data[1].valid := 1, [87].log_data[2].valid := 1, [87].log_data[3].valid := 1, [87].log_data[4].valid := 1, [87].log_data[5].valid := 1, [87].log_data[6].valid := 1, [87].log_data[7].valid := 1, [87].log_data[8].valid := 1, [87].log_data[9].valid := 1, [87].log_data[10].valid := 1, [87].log_data[11].valid := 1, [87].log_data[12].valid := 1, [87].log_data[13].valid := 1, [87].log_data[14].valid := 1, [87].log_data[15].valid := 1, [87].log_data[16].valid := 1, [87].log_data[17].valid := 1, [87].log_data[18].valid := 1, [87].log_data[19].valid := 1, [87].time.Year := 2023, [87].time.Month := 1, [87].time.Day := 18, [87].time.Hour := 7, [87].time.Minute := 39, [87].time.Second := 59, [88].log_data[0].min := 1.0, [88].log_data[0].max := 1.0, [88].log_data[0].total := 300.0, [88].log_data[0].time := 300.0, [88].log_data[0].minminute := 40, [88].log_data[0].maxminute := 40, [88].log_data[0].valid := 1, [88].log_data[1].valid := 1, [88].log_data[2].valid := 1, [88].log_data[3].valid := 1, [88].log_data[4].valid := 1, [88].log_data[5].valid := 1, [88].log_data[6].valid := 1, [88].log_data[7].valid := 1, [88].log_data[8].valid := 1, [88].log_data[9].valid := 1, [88].log_data[10].valid := 1, [88].log_data[11].valid := 1, [88].log_data[12].valid := 1, [88].log_data[13].valid := 1, [88].log_data[14].valid := 1, [88].log_data[15].valid := 1, [88].log_data[16].valid := 1, [88].log_data[17].valid := 1, [88].log_data[18].valid := 1, [88].log_data[19].valid := 1,
        [88].time.Year := 2023, [88].time.Month := 1, [88].time.Day := 18, [88].time.Hour := 7, [88].time.Minute := 44, [88].time.Second := 59, [89].log_data[0].min := 1.0, [89].log_data[0].max := 1.0, [89].log_data[0].total := 300.0, [89].log_data[0].time := 300.0, [89].log_data[0].minminute := 45, [89].log_data[0].maxminute := 45, [89].log_data[0].valid := 1, [89].log_data[1].valid := 1, [89].log_data[2].valid := 1, [89].log_data[3].valid := 1, [89].log_data[4].valid := 1, [89].log_data[5].valid := 1, [89].log_data[6].valid := 1, [89].log_data[7].valid := 1, [89].log_data[8].valid := 1, [89].log_data[9].valid := 1, [89].log_data[10].valid := 1, [89].log_data[11].valid := 1, [89].log_data[12].valid := 1, [89].log_data[13].valid := 1, [89].log_data[14].valid := 1, [89].log_data[15].valid := 1, [89].log_data[16].valid := 1, [89].log_data[17].valid := 1, [89].log_data[18].valid := 1, [89].log_data[19].valid := 1, [89].time.Year := 2023, [89].time.Month := 1, [89].time.Day := 18, [89].time.Hour := 7, [89].time.Minute := 49, [89].time.Second := 59, [90].log_data[0].min := 1.0, [90].log_data[0].max := 1.0, [90].log_data[0].total := 300.0, [90].log_data[0].time := 300.0, [90].log_data[0].minminute := 50, [90].log_data[0].maxminute := 50, [90].log_data[0].valid := 1, [90].log_data[1].valid := 1, [90].log_data[2].valid := 1, [90].log_data[3].valid := 1, [90].log_data[4].valid := 1, [90].log_data[5].valid := 1, [90].log_data[6].valid := 1, [90].log_data[7].valid := 1, [90].log_data[8].valid := 1, [90].log_data[9].valid := 1, [90].log_data[10].valid := 1, [90].log_data[11].valid := 1, [90].log_data[12].valid := 1, [90].log_data[13].valid := 1, [90].log_data[14].valid := 1, [90].log_data[15].valid := 1,
        [90].log_data[16].valid := 1, [90].log_data[17].valid := 1, [90].log_data[18].valid := 1, [90].log_data[19].valid := 1, [90].time.Year := 2023, [90].time.Month := 1, [90].time.Day := 18, [90].time.Hour := 7, [90].time.Minute := 54, [90].time.Second := 59, [91].log_data[0].min := 1.0, [91].log_data[0].max := 1.0, [91].log_data[0].total := 300.0, [91].log_data[0].time := 300.0, [91].log_data[0].minminute := 55, [91].log_data[0].maxminute := 55, [91].log_data[0].valid := 1, [91].log_data[1].valid := 1, [91].log_data[2].valid := 1, [91].log_data[3].valid := 1, [91].log_data[4].valid := 1, [91].log_data[5].valid := 1, [91].log_data[6].valid := 1, [91].log_data[7].valid := 1, [91].log_data[8].valid := 1, [91].log_data[9].valid := 1, [91].log_data[10].valid := 1, [91].log_data[11].valid := 1, [91].log_data[12].valid := 1, [91].log_data[13].valid := 1, [91].log_data[14].valid := 1, [91].log_data[15].valid := 1, [91].log_data[16].valid := 1, [91].log_data[17].valid := 1, [91].log_data[18].valid := 1, [91].log_data[19].valid := 1, [91].time.Year := 2023, [91].time.Month := 1, [91].time.Day := 18, [91].time.Hour := 7, [91].time.Minute := 59, [91].time.Second := 59, [92].log_data[0].min := 1.0, [92].log_data[0].max := 1.0, [92].log_data[0].total := 299.5, [92].log_data[0].time := 299.5, [92].log_data[0].valid := 1, [92].log_data[1].valid := 1, [92].log_data[2].valid := 1, [92].log_data[3].valid := 1, [92].log_data[4].valid := 1, [92].log_data[5].valid := 1, [92].log_data[6].valid := 1, [92].log_data[7].valid := 1, [92].log_data[8].valid := 1, [92].log_data[9].valid := 1, [92].log_data[10].valid := 1, [92].log_data[11].valid := 1, [92].log_data[12].valid := 1, [92].log_data[13].valid := 1,
        [92].log_data[14].valid := 1, [92].log_data[15].valid := 1, [92].log_data[16].valid := 1, [92].log_data[17].valid := 1, [92].log_data[18].valid := 1, [92].log_data[19].valid := 1, [92].time.Year := 2023, [92].time.Month := 1, [92].time.Day := 18, [92].time.Hour := 8, [92].time.Minute := 4, [92].time.Second := 59, [93].log_data[0].min := 1.0, [93].log_data[0].max := 1.0, [93].log_data[0].total := 300.0, [93].log_data[0].time := 300.0, [93].log_data[0].minminute := 5, [93].log_data[0].maxminute := 5, [93].log_data[0].valid := 1, [93].log_data[1].valid := 1, [93].log_data[2].valid := 1, [93].log_data[3].valid := 1, [93].log_data[4].valid := 1, [93].log_data[5].valid := 1, [93].log_data[6].valid := 1, [93].log_data[7].valid := 1, [93].log_data[8].valid := 1, [93].log_data[9].valid := 1, [93].log_data[10].valid := 1, [93].log_data[11].valid := 1, [93].log_data[12].valid := 1, [93].log_data[13].valid := 1, [93].log_data[14].valid := 1, [93].log_data[15].valid := 1, [93].log_data[16].valid := 1, [93].log_data[17].valid := 1, [93].log_data[18].valid := 1, [93].log_data[19].valid := 1, [93].time.Year := 2023, [93].time.Month := 1, [93].time.Day := 18, [93].time.Hour := 8, [93].time.Minute := 9, [93].time.Second := 59, [94].log_data[0].min := 1.0, [94].log_data[0].max := 1.0, [94].log_data[0].total := 300.0, [94].log_data[0].time := 300.0, [94].log_data[0].minminute := 10, [94].log_data[0].maxminute := 10, [94].log_data[0].valid := 1, [94].log_data[1].valid := 1, [94].log_data[2].valid := 1, [94].log_data[3].valid := 1, [94].log_data[4].valid := 1, [94].log_data[5].valid := 1, [94].log_data[6].valid := 1, [94].log_data[7].valid := 1, [94].log_data[8].valid := 1, [94].log_data[9].valid := 1,
        [94].log_data[10].valid := 1, [94].log_data[11].valid := 1, [94].log_data[12].valid := 1, [94].log_data[13].valid := 1, [94].log_data[14].valid := 1, [94].log_data[15].valid := 1, [94].log_data[16].valid := 1, [94].log_data[17].valid := 1, [94].log_data[18].valid := 1, [94].log_data[19].valid := 1, [94].time.Year := 2023, [94].time.Month := 1, [94].time.Day := 18, [94].time.Hour := 8, [94].time.Minute := 14, [94].time.Second := 59, [95].log_data[0].min := 1.0, [95].log_data[0].max := 1.0, [95].log_data[0].total := 300.0, [95].log_data[0].time := 300.0, [95].log_data[0].minminute := 15, [95].log_data[0].maxminute := 15, [95].log_data[0].valid := 1, [95].log_data[1].valid := 1, [95].log_data[2].valid := 1, [95].log_data[3].valid := 1, [95].log_data[4].valid := 1, [95].log_data[5].valid := 1, [95].log_data[6].valid := 1, [95].log_data[7].valid := 1, [95].log_data[8].valid := 1, [95].log_data[9].valid := 1, [95].log_data[10].valid := 1, [95].log_data[11].valid := 1, [95].log_data[12].valid := 1, [95].log_data[13].valid := 1, [95].log_data[14].valid := 1, [95].log_data[15].valid := 1, [95].log_data[16].valid := 1, [95].log_data[17].valid := 1, [95].log_data[18].valid := 1, [95].log_data[19].valid := 1, [95].time.Year := 2023, [95].time.Month := 1, [95].time.Day := 18, [95].time.Hour := 8, [95].time.Minute := 19, [95].time.Second := 59, [96].log_data[0].min := 1.0, [96].log_data[0].max := 1.0, [96].log_data[0].total := 300.0, [96].log_data[0].time := 300.0, [96].log_data[0].minminute := 20, [96].log_data[0].maxminute := 20, [96].log_data[0].valid := 1, [96].log_data[1].valid := 1, [96].log_data[2].valid := 1, [96].log_data[3].valid := 1, [96].log_data[4].valid := 1, [96].log_data[5].valid := 1,
        [96].log_data[6].valid := 1, [96].log_data[7].valid := 1, [96].log_data[8].valid := 1, [96].log_data[9].valid := 1, [96].log_data[10].valid := 1, [96].log_data[11].valid := 1, [96].log_data[12].valid := 1, [96].log_data[13].valid := 1, [96].log_data[14].valid := 1, [96].log_data[15].valid := 1, [96].log_data[16].valid := 1, [96].log_data[17].valid := 1, [96].log_data[18].valid := 1, [96].log_data[19].valid := 1, [96].time.Year := 2023, [96].time.Month := 1, [96].time.Day := 18, [96].time.Hour := 8, [96].time.Minute := 24, [96].time.Second := 59, [97].log_data[0].min := 1.0, [97].log_data[0].max := 1.0, [97].log_data[0].total := 300.0, [97].log_data[0].time := 300.0, [97].log_data[0].minminute := 25, [97].log_data[0].maxminute := 25, [97].log_data[0].valid := 1, [97].log_data[1].valid := 1, [97].log_data[2].valid := 1, [97].log_data[3].valid := 1, [97].log_data[4].valid := 1, [97].log_data[5].valid := 1, [97].log_data[6].valid := 1, [97].log_data[7].valid := 1, [97].log_data[8].valid := 1, [97].log_data[9].valid := 1, [97].log_data[10].valid := 1, [97].log_data[11].valid := 1, [97].log_data[12].valid := 1, [97].log_data[13].valid := 1, [97].log_data[14].valid := 1, [97].log_data[15].valid := 1, [97].log_data[16].valid := 1, [97].log_data[17].valid := 1, [97].log_data[18].valid := 1, [97].log_data[19].valid := 1, [97].time.Year := 2023, [97].time.Month := 1, [97].time.Day := 18, [97].time.Hour := 8, [97].time.Minute := 29, [97].time.Second := 59, [98].log_data[0].min := 1.0, [98].log_data[0].max := 1.0, [98].log_data[0].total := 300.0, [98].log_data[0].time := 300.0, [98].log_data[0].minminute := 30, [98].log_data[0].maxminute := 30, [98].log_data[0].valid := 1, [98].log_data[1].valid := 1,
        [98].log_data[2].valid := 1, [98].log_data[3].valid := 1, [98].log_data[4].valid := 1, [98].log_data[5].valid := 1, [98].log_data[6].valid := 1, [98].log_data[7].valid := 1, [98].log_data[8].valid := 1, [98].log_data[9].valid := 1, [98].log_data[10].valid := 1, [98].log_data[11].valid := 1, [98].log_data[12].valid := 1, [98].log_data[13].valid := 1, [98].log_data[14].valid := 1, [98].log_data[15].valid := 1, [98].log_data[16].valid := 1, [98].log_data[17].valid := 1, [98].log_data[18].valid := 1, [98].log_data[19].valid := 1, [98].time.Year := 2023, [98].time.Month := 1, [98].time.Day := 18, [98].time.Hour := 8, [98].time.Minute := 34, [98].time.Second := 59, [99].log_data[0].min := 1.0, [99].log_data[0].max := 1.0, [99].log_data[0].total := 300.0, [99].log_data[0].time := 300.0, [99].log_data[0].minminute := 35, [99].log_data[0].maxminute := 35, [99].log_data[0].valid := 1, [99].log_data[1].valid := 1, [99].log_data[2].valid := 1, [99].log_data[3].valid := 1, [99].log_data[4].valid := 1, [99].log_data[5].valid := 1, [99].log_data[6].valid := 1, [99].log_data[7].valid := 1, [99].log_data[8].valid := 1, [99].log_data[9].valid := 1, [99].log_data[10].valid := 1, [99].log_data[11].valid := 1, [99].log_data[12].valid := 1, [99].log_data[13].valid := 1, [99].log_data[14].valid := 1, [99].log_data[15].valid := 1, [99].log_data[16].valid := 1, [99].log_data[17].valid := 1, [99].log_data[18].valid := 1, [99].log_data[19].valid := 1, [99].time.Year := 2023, [99].time.Month := 1, [99].time.Day := 18, [99].time.Hour := 8, [99].time.Minute := 39, [99].time.Second := 59, [100].log_data[0].min := 1.0, [100].log_data[0].max := 1.0, [100].log_data[0].total := 300.0, [100].log_data[0].time := 300.0,
        [100].log_data[0].minminute := 40, [100].log_data[0].maxminute := 40, [100].log_data[0].valid := 1, [100].log_data[1].valid := 1, [100].log_data[2].valid := 1, [100].log_data[3].valid := 1, [100].log_data[4].valid := 1, [100].log_data[5].valid := 1, [100].log_data[6].valid := 1, [100].log_data[7].valid := 1, [100].log_data[8].valid := 1, [100].log_data[9].valid := 1, [100].log_data[10].valid := 1, [100].log_data[11].valid := 1, [100].log_data[12].valid := 1, [100].log_data[13].valid := 1, [100].log_data[14].valid := 1, [100].log_data[15].valid := 1, [100].log_data[16].valid := 1, [100].log_data[17].valid := 1, [100].log_data[18].valid := 1, [100].log_data[19].valid := 1, [100].time.Year := 2023, [100].time.Month := 1, [100].time.Day := 18, [100].time.Hour := 8, [100].time.Minute := 44, [100].time.Second := 59, [101].log_data[0].min := 1.0, [101].log_data[0].max := 1.0, [101].log_data[0].total := 300.0, [101].log_data[0].time := 300.0, [101].log_data[0].minminute := 45, [101].log_data[0].maxminute := 45, [101].log_data[0].valid := 1, [101].log_data[1].valid := 1, [101].log_data[2].valid := 1, [101].log_data[3].valid := 1, [101].log_data[4].valid := 1, [101].log_data[5].valid := 1, [101].log_data[6].valid := 1, [101].log_data[7].valid := 1, [101].log_data[8].valid := 1, [101].log_data[9].valid := 1, [101].log_data[10].valid := 1, [101].log_data[11].valid := 1, [101].log_data[12].valid := 1, [101].log_data[13].valid := 1, [101].log_data[14].valid := 1, [101].log_data[15].valid := 1, [101].log_data[16].valid := 1, [101].log_data[17].valid := 1, [101].log_data[18].valid := 1, [101].log_data[19].valid := 1, [101].time.Year := 2023, [101].time.Month := 1, [101].time.Day := 18, [101].time.Hour := 8, [101].time.Minute := 49, [101].time.Second := 59,
        [102].log_data[0].min := 1.0, [102].log_data[0].max := 1.0, [102].log_data[0].total := 300.0, [102].log_data[0].time := 300.0, [102].log_data[0].minminute := 50, [102].log_data[0].maxminute := 50, [102].log_data[0].valid := 1, [102].log_data[1].valid := 1, [102].log_data[2].valid := 1, [102].log_data[3].valid := 1, [102].log_data[4].valid := 1, [102].log_data[5].valid := 1, [102].log_data[6].valid := 1, [102].log_data[7].valid := 1, [102].log_data[8].valid := 1, [102].log_data[9].valid := 1, [102].log_data[10].valid := 1, [102].log_data[11].valid := 1, [102].log_data[12].valid := 1, [102].log_data[13].valid := 1, [102].log_data[14].valid := 1, [102].log_data[15].valid := 1, [102].log_data[16].valid := 1, [102].log_data[17].valid := 1, [102].log_data[18].valid := 1, [102].log_data[19].valid := 1, [102].time.Year := 2023, [102].time.Month := 1, [102].time.Day := 18, [102].time.Hour := 8, [102].time.Minute := 54, [102].time.Second := 59, [103].log_data[0].min := 1.0, [103].log_data[0].max := 1.0, [103].log_data[0].total := 300.0, [103].log_data[0].time := 300.0, [103].log_data[0].minminute := 55, [103].log_data[0].maxminute := 55, [103].log_data[0].valid := 1, [103].log_data[1].valid := 1, [103].log_data[2].valid := 1, [103].log_data[3].valid := 1, [103].log_data[4].valid := 1, [103].log_data[5].valid := 1, [103].log_data[6].valid := 1, [103].log_data[7].valid := 1, [103].log_data[8].valid := 1, [103].log_data[9].valid := 1, [103].log_data[10].valid := 1, [103].log_data[11].valid := 1, [103].log_data[12].valid := 1, [103].log_data[13].valid := 1, [103].log_data[14].valid := 1, [103].log_data[15].valid := 1, [103].log_data[16].valid := 1, [103].log_data[17].valid := 1, [103].log_data[18].valid := 1, [103].log_data[19].valid := 1, [103].time.Year := 2023, [103].time.Month := 1,
        [103].time.Day := 18, [103].time.Hour := 8, [103].time.Minute := 59, [103].time.Second := 59, [104].log_data[0].min := 1.0, [104].log_data[0].max := 1.0, [104].log_data[0].total := 300.0, [104].log_data[0].time := 300.0, [104].log_data[0].valid := 1, [104].log_data[1].valid := 1, [104].log_data[2].valid := 1, [104].log_data[3].valid := 1, [104].log_data[4].valid := 1, [104].log_data[5].valid := 1, [104].log_data[6].valid := 1, [104].log_data[7].valid := 1, [104].log_data[8].valid := 1, [104].log_data[9].valid := 1, [104].log_data[10].valid := 1, [104].log_data[11].valid := 1, [104].log_data[12].valid := 1, [104].log_data[13].valid := 1, [104].log_data[14].valid := 1, [104].log_data[15].valid := 1, [104].log_data[16].valid := 1, [104].log_data[17].valid := 1, [104].log_data[18].valid := 1, [104].log_data[19].valid := 1, [104].time.Year := 2023, [104].time.Month := 1, [104].time.Day := 18, [104].time.Hour := 9, [104].time.Minute := 4, [104].time.Second := 59, [105].log_data[0].min := 1.0, [105].log_data[0].max := 1.0, [105].log_data[0].total := 300.0, [105].log_data[0].time := 300.0, [105].log_data[0].minminute := 5, [105].log_data[0].maxminute := 5, [105].log_data[0].valid := 1, [105].log_data[1].valid := 1, [105].log_data[2].valid := 1, [105].log_data[3].valid := 1, [105].log_data[4].valid := 1, [105].log_data[5].valid := 1, [105].log_data[6].valid := 1, [105].log_data[7].valid := 1, [105].log_data[8].valid := 1, [105].log_data[9].valid := 1, [105].log_data[10].valid := 1, [105].log_data[11].valid := 1, [105].log_data[12].valid := 1, [105].log_data[13].valid := 1, [105].log_data[14].valid := 1, [105].log_data[15].valid := 1, [105].log_data[16].valid := 1, [105].log_data[17].valid := 1, [105].log_data[18].valid := 1, [105].log_data[19].valid := 1,
        [105].time.Year := 2023, [105].time.Month := 1, [105].time.Day := 18, [105].time.Hour := 9, [105].time.Minute := 9, [105].time.Second := 59, [106].log_data[0].min := 1.0, [106].log_data[0].max := 1.0, [106].log_data[0].total := 300.0, [106].log_data[0].time := 300.0, [106].log_data[0].minminute := 10, [106].log_data[0].maxminute := 10, [106].log_data[0].valid := 1, [106].log_data[1].valid := 1, [106].log_data[2].valid := 1, [106].log_data[3].valid := 1, [106].log_data[4].valid := 1, [106].log_data[5].valid := 1, [106].log_data[6].valid := 1, [106].log_data[7].valid := 1, [106].log_data[8].valid := 1, [106].log_data[9].valid := 1, [106].log_data[10].valid := 1, [106].log_data[11].valid := 1, [106].log_data[12].valid := 1, [106].log_data[13].valid := 1, [106].log_data[14].valid := 1, [106].log_data[15].valid := 1, [106].log_data[16].valid := 1, [106].log_data[17].valid := 1, [106].log_data[18].valid := 1, [106].log_data[19].valid := 1, [106].time.Year := 2023, [106].time.Month := 1, [106].time.Day := 18, [106].time.Hour := 9, [106].time.Minute := 14, [106].time.Second := 59, [107].log_data[0].min := 1.0, [107].log_data[0].max := 1.0, [107].log_data[0].total := 300.0, [107].log_data[0].time := 300.0, [107].log_data[0].minminute := 15, [107].log_data[0].maxminute := 15, [107].log_data[0].valid := 1, [107].log_data[1].valid := 1, [107].log_data[2].valid := 1, [107].log_data[3].valid := 1, [107].log_data[4].valid := 1, [107].log_data[5].valid := 1, [107].log_data[6].valid := 1, [107].log_data[7].valid := 1, [107].log_data[8].valid := 1, [107].log_data[9].valid := 1, [107].log_data[10].valid := 1, [107].log_data[11].valid := 1, [107].log_data[12].valid := 1, [107].log_data[13].valid := 1, [107].log_data[14].valid := 1, [107].log_data[15].valid := 1,
        [107].log_data[16].valid := 1, [107].log_data[17].valid := 1, [107].log_data[18].valid := 1, [107].log_data[19].valid := 1, [107].time.Year := 2023, [107].time.Month := 1, [107].time.Day := 18, [107].time.Hour := 9, [107].time.Minute := 19, [107].time.Second := 59, [108].log_data[0].min := 1.0, [108].log_data[0].max := 1.0, [108].log_data[0].total := 300.0, [108].log_data[0].time := 300.0, [108].log_data[0].minminute := 20, [108].log_data[0].maxminute := 20, [108].log_data[0].valid := 1, [108].log_data[1].valid := 1, [108].log_data[2].valid := 1, [108].log_data[3].valid := 1, [108].log_data[4].valid := 1, [108].log_data[5].valid := 1, [108].log_data[6].valid := 1, [108].log_data[7].valid := 1, [108].log_data[8].valid := 1, [108].log_data[9].valid := 1, [108].log_data[10].valid := 1, [108].log_data[11].valid := 1, [108].log_data[12].valid := 1, [108].log_data[13].valid := 1, [108].log_data[14].valid := 1, [108].log_data[15].valid := 1, [108].log_data[16].valid := 1, [108].log_data[17].valid := 1, [108].log_data[18].valid := 1, [108].log_data[19].valid := 1, [108].time.Year := 2023, [108].time.Month := 1, [108].time.Day := 18, [108].time.Hour := 9, [108].time.Minute := 24, [108].time.Second := 59, [109].log_data[0].min := 1.0, [109].log_data[0].max := 1.0, [109].log_data[0].total := 300.0, [109].log_data[0].time := 300.0, [109].log_data[0].minminute := 25, [109].log_data[0].maxminute := 25, [109].log_data[0].valid := 1, [109].log_data[1].valid := 1, [109].log_data[2].valid := 1, [109].log_data[3].valid := 1, [109].log_data[4].valid := 1, [109].log_data[5].valid := 1, [109].log_data[6].valid := 1, [109].log_data[7].valid := 1, [109].log_data[8].valid := 1, [109].log_data[9].valid := 1, [109].log_data[10].valid := 1, [109].log_data[11].valid := 1,
        [109].log_data[12].valid := 1, [109].log_data[13].valid := 1, [109].log_data[14].valid := 1, [109].log_data[15].valid := 1, [109].log_data[16].valid := 1, [109].log_data[17].valid := 1, [109].log_data[18].valid := 1, [109].log_data[19].valid := 1, [109].time.Year := 2023, [109].time.Month := 1, [109].time.Day := 18, [109].time.Hour := 9, [109].time.Minute := 29, [109].time.Second := 59, [110].log_data[0].min := 1.0, [110].log_data[0].max := 1.0, [110].log_data[0].total := 300.0, [110].log_data[0].time := 300.0, [110].log_data[0].minminute := 30, [110].log_data[0].maxminute := 30, [110].log_data[0].valid := 1, [110].log_data[1].valid := 1, [110].log_data[2].valid := 1, [110].log_data[3].valid := 1, [110].log_data[4].valid := 1, [110].log_data[5].valid := 1, [110].log_data[6].valid := 1, [110].log_data[7].valid := 1, [110].log_data[8].valid := 1, [110].log_data[9].valid := 1, [110].log_data[10].valid := 1, [110].log_data[11].valid := 1, [110].log_data[12].valid := 1, [110].log_data[13].valid := 1, [110].log_data[14].valid := 1, [110].log_data[15].valid := 1, [110].log_data[16].valid := 1, [110].log_data[17].valid := 1, [110].log_data[18].valid := 1, [110].log_data[19].valid := 1, [110].time.Year := 2023, [110].time.Month := 1, [110].time.Day := 18, [110].time.Hour := 9, [110].time.Minute := 34, [110].time.Second := 59, [111].log_data[0].min := 1.0, [111].log_data[0].max := 1.0, [111].log_data[0].total := 300.0, [111].log_data[0].time := 300.0, [111].log_data[0].minminute := 35, [111].log_data[0].maxminute := 35, [111].log_data[0].valid := 1, [111].log_data[1].valid := 1, [111].log_data[2].valid := 1, [111].log_data[3].valid := 1, [111].log_data[4].valid := 1, [111].log_data[5].valid := 1, [111].log_data[6].valid := 1, [111].log_data[7].valid := 1,
        [111].log_data[8].valid := 1, [111].log_data[9].valid := 1, [111].log_data[10].valid := 1, [111].log_data[11].valid := 1, [111].log_data[12].valid := 1, [111].log_data[13].valid := 1, [111].log_data[14].valid := 1, [111].log_data[15].valid := 1, [111].log_data[16].valid := 1, [111].log_data[17].valid := 1, [111].log_data[18].valid := 1, [111].log_data[19].valid := 1, [111].time.Year := 2023, [111].time.Month := 1, [111].time.Day := 18, [111].time.Hour := 9, [111].time.Minute := 39, [111].time.Second := 59, [112].log_data[0].min := 1.0, [112].log_data[0].max := 1.0, [112].log_data[0].total := 300.0, [112].log_data[0].time := 300.0, [112].log_data[0].minminute := 40, [112].log_data[0].maxminute := 40, [112].log_data[0].valid := 1, [112].log_data[1].valid := 1, [112].log_data[2].valid := 1, [112].log_data[3].valid := 1, [112].log_data[4].valid := 1, [112].log_data[5].valid := 1, [112].log_data[6].valid := 1, [112].log_data[7].valid := 1, [112].log_data[8].valid := 1, [112].log_data[9].valid := 1, [112].log_data[10].valid := 1, [112].log_data[11].valid := 1, [112].log_data[12].valid := 1, [112].log_data[13].valid := 1, [112].log_data[14].valid := 1, [112].log_data[15].valid := 1, [112].log_data[16].valid := 1, [112].log_data[17].valid := 1, [112].log_data[18].valid := 1, [112].log_data[19].valid := 1, [112].time.Year := 2023, [112].time.Month := 1, [112].time.Day := 18, [112].time.Hour := 9, [112].time.Minute := 44, [112].time.Second := 59, [113].log_data[0].min := 1.0, [113].log_data[0].max := 1.0, [113].log_data[0].total := 300.0, [113].log_data[0].time := 300.0, [113].log_data[0].minminute := 45, [113].log_data[0].maxminute := 45, [113].log_data[0].valid := 1, [113].log_data[1].valid := 1, [113].log_data[2].valid := 1, [113].log_data[3].valid := 1,
        [113].log_data[4].valid := 1, [113].log_data[5].valid := 1, [113].log_data[6].valid := 1, [113].log_data[7].valid := 1, [113].log_data[8].valid := 1, [113].log_data[9].valid := 1, [113].log_data[10].valid := 1, [113].log_data[11].valid := 1, [113].log_data[12].valid := 1, [113].log_data[13].valid := 1, [113].log_data[14].valid := 1, [113].log_data[15].valid := 1, [113].log_data[16].valid := 1, [113].log_data[17].valid := 1, [113].log_data[18].valid := 1, [113].log_data[19].valid := 1, [113].time.Year := 2023, [113].time.Month := 1, [113].time.Day := 18, [113].time.Hour := 9, [113].time.Minute := 49, [113].time.Second := 59, [114].log_data[0].min := 1.0, [114].log_data[0].max := 1.0, [114].log_data[0].total := 300.0, [114].log_data[0].time := 300.0, [114].log_data[0].minminute := 50, [114].log_data[0].maxminute := 50, [114].log_data[0].valid := 1, [114].log_data[1].valid := 1, [114].log_data[2].valid := 1, [114].log_data[3].valid := 1, [114].log_data[4].valid := 1, [114].log_data[5].valid := 1, [114].log_data[6].valid := 1, [114].log_data[7].valid := 1, [114].log_data[8].valid := 1, [114].log_data[9].valid := 1, [114].log_data[10].valid := 1, [114].log_data[11].valid := 1, [114].log_data[12].valid := 1, [114].log_data[13].valid := 1, [114].log_data[14].valid := 1, [114].log_data[15].valid := 1, [114].log_data[16].valid := 1, [114].log_data[17].valid := 1, [114].log_data[18].valid := 1, [114].log_data[19].valid := 1, [114].time.Year := 2023, [114].time.Month := 1, [114].time.Day := 18, [114].time.Hour := 9, [114].time.Minute := 54, [114].time.Second := 59, [115].log_data[0].min := 1.0, [115].log_data[0].max := 1.0, [115].log_data[0].total := 300.0, [115].log_data[0].time := 300.0, [115].log_data[0].minminute := 55, [115].log_data[0].maxminute := 55,
        [115].log_data[0].valid := 1, [115].log_data[1].valid := 1, [115].log_data[2].valid := 1, [115].log_data[3].valid := 1, [115].log_data[4].valid := 1, [115].log_data[5].valid := 1, [115].log_data[6].valid := 1, [115].log_data[7].valid := 1, [115].log_data[8].valid := 1, [115].log_data[9].valid := 1, [115].log_data[10].valid := 1, [115].log_data[11].valid := 1, [115].log_data[12].valid := 1, [115].log_data[13].valid := 1, [115].log_data[14].valid := 1, [115].log_data[15].valid := 1, [115].log_data[16].valid := 1, [115].log_data[17].valid := 1, [115].log_data[18].valid := 1, [115].log_data[19].valid := 1, [115].time.Year := 2023, [115].time.Month := 1, [115].time.Day := 18, [115].time.Hour := 9, [115].time.Minute := 59, [115].time.Second := 59, [116].log_data[0].min := 1.0, [116].log_data[0].max := 1.0, [116].log_data[0].total := 300.0, [116].log_data[0].time := 300.0, [116].log_data[0].valid := 1, [116].log_data[1].valid := 1, [116].log_data[2].valid := 1, [116].log_data[3].valid := 1, [116].log_data[4].valid := 1, [116].log_data[5].valid := 1, [116].log_data[6].valid := 1, [116].log_data[7].valid := 1, [116].log_data[8].valid := 1, [116].log_data[9].valid := 1, [116].log_data[10].valid := 1, [116].log_data[11].valid := 1, [116].log_data[12].valid := 1, [116].log_data[13].valid := 1, [116].log_data[14].valid := 1, [116].log_data[15].valid := 1, [116].log_data[16].valid := 1, [116].log_data[17].valid := 1, [116].log_data[18].valid := 1, [116].log_data[19].valid := 1, [116].time.Year := 2023, [116].time.Month := 1, [116].time.Day := 18, [116].time.Hour := 10, [116].time.Minute := 4, [116].time.Second := 59, [117].log_data[0].min := 1.0, [117].log_data[0].max := 1.0, [117].log_data[0].total := 300.0, [117].log_data[0].time := 300.0,
        [117].log_data[0].minminute := 5, [117].log_data[0].maxminute := 5, [117].log_data[0].valid := 1, [117].log_data[1].valid := 1, [117].log_data[2].valid := 1, [117].log_data[3].valid := 1, [117].log_data[4].valid := 1, [117].log_data[5].valid := 1, [117].log_data[6].valid := 1, [117].log_data[7].valid := 1, [117].log_data[8].valid := 1, [117].log_data[9].valid := 1, [117].log_data[10].valid := 1, [117].log_data[11].valid := 1, [117].log_data[12].valid := 1, [117].log_data[13].valid := 1, [117].log_data[14].valid := 1, [117].log_data[15].valid := 1, [117].log_data[16].valid := 1, [117].log_data[17].valid := 1, [117].log_data[18].valid := 1, [117].log_data[19].valid := 1, [117].time.Year := 2023, [117].time.Month := 1, [117].time.Day := 18, [117].time.Hour := 10, [117].time.Minute := 9, [117].time.Second := 59, [118].log_data[0].min := 1.0, [118].log_data[0].max := 1.0, [118].log_data[0].total := 300.0, [118].log_data[0].time := 300.0, [118].log_data[0].minminute := 10, [118].log_data[0].maxminute := 10, [118].log_data[0].valid := 1, [118].log_data[1].valid := 1, [118].log_data[2].valid := 1, [118].log_data[3].valid := 1, [118].log_data[4].valid := 1, [118].log_data[5].valid := 1, [118].log_data[6].valid := 1, [118].log_data[7].valid := 1, [118].log_data[8].valid := 1, [118].log_data[9].valid := 1, [118].log_data[10].valid := 1, [118].log_data[11].valid := 1, [118].log_data[12].valid := 1, [118].log_data[13].valid := 1, [118].log_data[14].valid := 1, [118].log_data[15].valid := 1, [118].log_data[16].valid := 1, [118].log_data[17].valid := 1, [118].log_data[18].valid := 1, [118].log_data[19].valid := 1, [118].time.Year := 2023, [118].time.Month := 1, [118].time.Day := 18, [118].time.Hour := 10, [118].time.Minute := 14, [118].time.Second := 59,
        [119].log_data[0].min := 1.0, [119].log_data[0].max := 1.0, [119].log_data[0].total := 300.0, [119].log_data[0].time := 300.0, [119].log_data[0].minminute := 15, [119].log_data[0].maxminute := 15, [119].log_data[0].valid := 1, [119].log_data[1].valid := 1, [119].log_data[2].valid := 1, [119].log_data[3].valid := 1, [119].log_data[4].valid := 1, [119].log_data[5].valid := 1, [119].log_data[6].valid := 1, [119].log_data[7].valid := 1, [119].log_data[8].valid := 1, [119].log_data[9].valid := 1, [119].log_data[10].valid := 1, [119].log_data[11].valid := 1, [119].log_data[12].valid := 1, [119].log_data[13].valid := 1, [119].log_data[14].valid := 1, [119].log_data[15].valid := 1, [119].log_data[16].valid := 1, [119].log_data[17].valid := 1, [119].log_data[18].valid := 1, [119].log_data[19].valid := 1, [119].time.Year := 2023, [119].time.Month := 1, [119].time.Day := 18, [119].time.Hour := 10, [119].time.Minute := 19, [119].time.Second := 59, [120].log_data[0].min := 1.0, [120].log_data[0].max := 1.0, [120].log_data[0].total := 300.0, [120].log_data[0].time := 300.0, [120].log_data[0].minminute := 20, [120].log_data[0].maxminute := 20, [120].log_data[0].valid := 1, [120].log_data[1].valid := 1, [120].log_data[2].valid := 1, [120].log_data[3].valid := 1, [120].log_data[4].valid := 1, [120].log_data[5].valid := 1, [120].log_data[6].valid := 1, [120].log_data[7].valid := 1, [120].log_data[8].valid := 1, [120].log_data[9].valid := 1, [120].log_data[10].valid := 1, [120].log_data[11].valid := 1, [120].log_data[12].valid := 1, [120].log_data[13].valid := 1, [120].log_data[14].valid := 1, [120].log_data[15].valid := 1, [120].log_data[16].valid := 1, [120].log_data[17].valid := 1, [120].log_data[18].valid := 1, [120].log_data[19].valid := 1, [120].time.Year := 2023, [120].time.Month := 1,
        [120].time.Day := 18, [120].time.Hour := 10, [120].time.Minute := 24, [120].time.Second := 59, [121].log_data[0].min := 1.0, [121].log_data[0].max := 1.0, [121].log_data[0].total := 300.0, [121].log_data[0].time := 300.0, [121].log_data[0].minminute := 25, [121].log_data[0].maxminute := 25, [121].log_data[0].valid := 1, [121].log_data[1].valid := 1, [121].log_data[2].valid := 1, [121].log_data[3].valid := 1, [121].log_data[4].valid := 1, [121].log_data[5].valid := 1, [121].log_data[6].valid := 1, [121].log_data[7].valid := 1, [121].log_data[8].valid := 1, [121].log_data[9].valid := 1, [121].log_data[10].valid := 1, [121].log_data[11].valid := 1, [121].log_data[12].valid := 1, [121].log_data[13].valid := 1, [121].log_data[14].valid := 1, [121].log_data[15].valid := 1, [121].log_data[16].valid := 1, [121].log_data[17].valid := 1, [121].log_data[18].valid := 1, [121].log_data[19].valid := 1, [121].time.Year := 2023, [121].time.Month := 1, [121].time.Day := 18, [121].time.Hour := 10, [121].time.Minute := 29, [121].time.Second := 59, [122].log_data[0].min := 1.0, [122].log_data[0].max := 1.0, [122].log_data[0].total := 300.0, [122].log_data[0].time := 300.0, [122].log_data[0].minminute := 30, [122].log_data[0].maxminute := 30, [122].log_data[0].valid := 1, [122].log_data[1].valid := 1, [122].log_data[2].valid := 1, [122].log_data[3].valid := 1, [122].log_data[4].valid := 1, [122].log_data[5].valid := 1, [122].log_data[6].valid := 1, [122].log_data[7].valid := 1, [122].log_data[8].valid := 1, [122].log_data[9].valid := 1, [122].log_data[10].valid := 1, [122].log_data[11].valid := 1, [122].log_data[12].valid := 1, [122].log_data[13].valid := 1, [122].log_data[14].valid := 1, [122].log_data[15].valid := 1, [122].log_data[16].valid := 1, [122].log_data[17].valid := 1,
        [122].log_data[18].valid := 1, [122].log_data[19].valid := 1, [122].time.Year := 2023, [122].time.Month := 1, [122].time.Day := 18, [122].time.Hour := 10, [122].time.Minute := 34, [122].time.Second := 59, [123].log_data[0].min := 1.0, [123].log_data[0].max := 1.0, [123].log_data[0].total := 300.0, [123].log_data[0].time := 300.0, [123].log_data[0].minminute := 35, [123].log_data[0].maxminute := 35, [123].log_data[0].valid := 1, [123].log_data[1].valid := 1, [123].log_data[2].valid := 1, [123].log_data[3].valid := 1, [123].log_data[4].valid := 1, [123].log_data[5].valid := 1, [123].log_data[6].valid := 1, [123].log_data[7].valid := 1, [123].log_data[8].valid := 1, [123].log_data[9].valid := 1, [123].log_data[10].valid := 1, [123].log_data[11].valid := 1, [123].log_data[12].valid := 1, [123].log_data[13].valid := 1, [123].log_data[14].valid := 1, [123].log_data[15].valid := 1, [123].log_data[16].valid := 1, [123].log_data[17].valid := 1, [123].log_data[18].valid := 1, [123].log_data[19].valid := 1, [123].time.Year := 2023, [123].time.Month := 1, [123].time.Day := 18, [123].time.Hour := 10, [123].time.Minute := 39, [123].time.Second := 59, [124].log_data[0].min := 1.0, [124].log_data[0].max := 1.0, [124].log_data[0].total := 300.0, [124].log_data[0].time := 300.0, [124].log_data[0].minminute := 40, [124].log_data[0].maxminute := 40, [124].log_data[0].valid := 1, [124].log_data[1].valid := 1, [124].log_data[2].valid := 1, [124].log_data[3].valid := 1, [124].log_data[4].valid := 1, [124].log_data[5].valid := 1, [124].log_data[6].valid := 1, [124].log_data[7].valid := 1, [124].log_data[8].valid := 1, [124].log_data[9].valid := 1, [124].log_data[10].valid := 1, [124].log_data[11].valid := 1, [124].log_data[12].valid := 1, [124].log_data[13].valid := 1,
        [124].log_data[14].valid := 1, [124].log_data[15].valid := 1, [124].log_data[16].valid := 1, [124].log_data[17].valid := 1, [124].log_data[18].valid := 1, [124].log_data[19].valid := 1, [124].time.Year := 2023, [124].time.Month := 1, [124].time.Day := 18, [124].time.Hour := 10, [124].time.Minute := 44, [124].time.Second := 59, [125].log_data[0].min := 1.0, [125].log_data[0].max := 1.0, [125].log_data[0].total := 300.0, [125].log_data[0].time := 300.0, [125].log_data[0].minminute := 45, [125].log_data[0].maxminute := 45, [125].log_data[0].valid := 1, [125].log_data[1].valid := 1, [125].log_data[2].valid := 1, [125].log_data[3].valid := 1, [125].log_data[4].valid := 1, [125].log_data[5].valid := 1, [125].log_data[6].valid := 1, [125].log_data[7].valid := 1, [125].log_data[8].valid := 1, [125].log_data[9].valid := 1, [125].log_data[10].valid := 1, [125].log_data[11].valid := 1, [125].log_data[12].valid := 1, [125].log_data[13].valid := 1, [125].log_data[14].valid := 1, [125].log_data[15].valid := 1, [125].log_data[16].valid := 1, [125].log_data[17].valid := 1, [125].log_data[18].valid := 1, [125].log_data[19].valid := 1, [125].time.Year := 2023, [125].time.Month := 1, [125].time.Day := 18, [125].time.Hour := 10, [125].time.Minute := 49, [125].time.Second := 59, [126].log_data[0].min := 1.0, [126].log_data[0].max := 1.0, [126].log_data[0].total := 300.0, [126].log_data[0].time := 300.0, [126].log_data[0].minminute := 50, [126].log_data[0].maxminute := 50, [126].log_data[0].valid := 1, [126].log_data[1].valid := 1, [126].log_data[2].valid := 1, [126].log_data[3].valid := 1, [126].log_data[4].valid := 1, [126].log_data[5].valid := 1, [126].log_data[6].valid := 1, [126].log_data[7].valid := 1, [126].log_data[8].valid := 1, [126].log_data[9].valid := 1,
        [126].log_data[10].valid := 1, [126].log_data[11].valid := 1, [126].log_data[12].valid := 1, [126].log_data[13].valid := 1, [126].log_data[14].valid := 1, [126].log_data[15].valid := 1, [126].log_data[16].valid := 1, [126].log_data[17].valid := 1, [126].log_data[18].valid := 1, [126].log_data[19].valid := 1, [126].time.Year := 2023, [126].time.Month := 1, [126].time.Day := 18, [126].time.Hour := 10, [126].time.Minute := 54, [126].time.Second := 59, [127].log_data[0].min := 1.0, [127].log_data[0].max := 1.0, [127].log_data[0].total := 300.0, [127].log_data[0].time := 300.0, [127].log_data[0].minminute := 55, [127].log_data[0].maxminute := 55, [127].log_data[0].valid := 1, [127].log_data[1].valid := 1, [127].log_data[2].valid := 1, [127].log_data[3].valid := 1, [127].log_data[4].valid := 1, [127].log_data[5].valid := 1, [127].log_data[6].valid := 1, [127].log_data[7].valid := 1, [127].log_data[8].valid := 1, [127].log_data[9].valid := 1, [127].log_data[10].valid := 1, [127].log_data[11].valid := 1, [127].log_data[12].valid := 1, [127].log_data[13].valid := 1, [127].log_data[14].valid := 1, [127].log_data[15].valid := 1, [127].log_data[16].valid := 1, [127].log_data[17].valid := 1, [127].log_data[18].valid := 1, [127].log_data[19].valid := 1, [127].time.Year := 2023, [127].time.Month := 1, [127].time.Day := 18, [127].time.Hour := 10, [127].time.Minute := 59, [127].time.Second := 59, [128].log_data[0].min := 1.0, [128].log_data[0].max := 1.0, [128].log_data[0].total := 300.0, [128].log_data[0].time := 300.0, [128].log_data[0].valid := 1, [128].log_data[1].valid := 1, [128].log_data[2].valid := 1, [128].log_data[3].valid := 1, [128].log_data[4].valid := 1, [128].log_data[5].valid := 1, [128].log_data[6].valid := 1, [128].log_data[7].valid := 1,
        [128].log_data[8].valid := 1, [128].log_data[9].valid := 1, [128].log_data[10].valid := 1, [128].log_data[11].valid := 1, [128].log_data[12].valid := 1, [128].log_data[13].valid := 1, [128].log_data[14].valid := 1, [128].log_data[15].valid := 1, [128].log_data[16].valid := 1, [128].log_data[17].valid := 1, [128].log_data[18].valid := 1, [128].log_data[19].valid := 1, [128].time.Year := 2023, [128].time.Month := 1, [128].time.Day := 18, [128].time.Hour := 11, [128].time.Minute := 4, [128].time.Second := 59, [129].log_data[0].min := 1.0, [129].log_data[0].max := 1.0, [129].log_data[0].total := 300.0, [129].log_data[0].time := 300.0, [129].log_data[0].minminute := 5, [129].log_data[0].maxminute := 5, [129].log_data[0].valid := 1, [129].log_data[1].valid := 1, [129].log_data[2].valid := 1, [129].log_data[3].valid := 1, [129].log_data[4].valid := 1, [129].log_data[5].valid := 1, [129].log_data[6].valid := 1, [129].log_data[7].valid := 1, [129].log_data[8].valid := 1, [129].log_data[9].valid := 1, [129].log_data[10].valid := 1, [129].log_data[11].valid := 1, [129].log_data[12].valid := 1, [129].log_data[13].valid := 1, [129].log_data[14].valid := 1, [129].log_data[15].valid := 1, [129].log_data[16].valid := 1, [129].log_data[17].valid := 1, [129].log_data[18].valid := 1, [129].log_data[19].valid := 1, [129].time.Year := 2023, [129].time.Month := 1, [129].time.Day := 18, [129].time.Hour := 11, [129].time.Minute := 9, [129].time.Second := 59, [130].log_data[0].min := 1.0, [130].log_data[0].max := 1.0, [130].log_data[0].total := 300.0, [130].log_data[0].time := 300.0, [130].log_data[0].minminute := 10, [130].log_data[0].maxminute := 10, [130].log_data[0].valid := 1, [130].log_data[1].valid := 1, [130].log_data[2].valid := 1, [130].log_data[3].valid := 1,
        [130].log_data[4].valid := 1, [130].log_data[5].valid := 1, [130].log_data[6].valid := 1, [130].log_data[7].valid := 1, [130].log_data[8].valid := 1, [130].log_data[9].valid := 1, [130].log_data[10].valid := 1, [130].log_data[11].valid := 1, [130].log_data[12].valid := 1, [130].log_data[13].valid := 1, [130].log_data[14].valid := 1, [130].log_data[15].valid := 1, [130].log_data[16].valid := 1, [130].log_data[17].valid := 1, [130].log_data[18].valid := 1, [130].log_data[19].valid := 1, [130].time.Year := 2023, [130].time.Month := 1, [130].time.Day := 18, [130].time.Hour := 11, [130].time.Minute := 14, [130].time.Second := 59, [131].log_data[0].min := 1.0, [131].log_data[0].max := 1.0, [131].log_data[0].total := 300.0, [131].log_data[0].time := 300.0, [131].log_data[0].minminute := 15, [131].log_data[0].maxminute := 15, [131].log_data[0].valid := 1, [131].log_data[1].valid := 1, [131].log_data[2].valid := 1, [131].log_data[3].valid := 1, [131].log_data[4].valid := 1, [131].log_data[5].valid := 1, [131].log_data[6].valid := 1, [131].log_data[7].valid := 1, [131].log_data[8].valid := 1, [131].log_data[9].valid := 1, [131].log_data[10].valid := 1, [131].log_data[11].valid := 1, [131].log_data[12].valid := 1, [131].log_data[13].valid := 1, [131].log_data[14].valid := 1, [131].log_data[15].valid := 1, [131].log_data[16].valid := 1, [131].log_data[17].valid := 1, [131].log_data[18].valid := 1, [131].log_data[19].valid := 1, [131].time.Year := 2023, [131].time.Month := 1, [131].time.Day := 18, [131].time.Hour := 11, [131].time.Minute := 19, [131].time.Second := 59, [132].log_data[0].min := 1.0, [132].log_data[0].max := 1.0, [132].log_data[0].total := 300.0, [132].log_data[0].time := 300.0, [132].log_data[0].minminute := 20, [132].log_data[0].maxminute := 20,
        [132].log_data[0].valid := 1, [132].log_data[1].valid := 1, [132].log_data[2].valid := 1, [132].log_data[3].valid := 1, [132].log_data[4].valid := 1, [132].log_data[5].valid := 1, [132].log_data[6].valid := 1, [132].log_data[7].valid := 1, [132].log_data[8].valid := 1, [132].log_data[9].valid := 1, [132].log_data[10].valid := 1, [132].log_data[11].valid := 1, [132].log_data[12].valid := 1, [132].log_data[13].valid := 1, [132].log_data[14].valid := 1, [132].log_data[15].valid := 1, [132].log_data[16].valid := 1, [132].log_data[17].valid := 1, [132].log_data[18].valid := 1, [132].log_data[19].valid := 1, [132].time.Year := 2023, [132].time.Month := 1, [132].time.Day := 18, [132].time.Hour := 11, [132].time.Minute := 24, [132].time.Second := 59, [133].log_data[0].min := 1.0, [133].log_data[0].max := 1.0, [133].log_data[0].total := 300.0, [133].log_data[0].time := 300.0, [133].log_data[0].minminute := 25, [133].log_data[0].maxminute := 25, [133].log_data[0].valid := 1, [133].log_data[1].valid := 1, [133].log_data[2].valid := 1, [133].log_data[3].valid := 1, [133].log_data[4].valid := 1, [133].log_data[5].valid := 1, [133].log_data[6].valid := 1, [133].log_data[7].valid := 1, [133].log_data[8].valid := 1, [133].log_data[9].valid := 1, [133].log_data[10].valid := 1, [133].log_data[11].valid := 1, [133].log_data[12].valid := 1, [133].log_data[13].valid := 1, [133].log_data[14].valid := 1, [133].log_data[15].valid := 1, [133].log_data[16].valid := 1, [133].log_data[17].valid := 1, [133].log_data[18].valid := 1, [133].log_data[19].valid := 1, [133].time.Year := 2023, [133].time.Month := 1, [133].time.Day := 18, [133].time.Hour := 11, [133].time.Minute := 29, [133].time.Second := 59, [134].log_data[0].min := 1.0, [134].log_data[0].max := 1.0,
        [134].log_data[0].total := 300.0, [134].log_data[0].time := 300.0, [134].log_data[0].minminute := 30, [134].log_data[0].maxminute := 30, [134].log_data[0].valid := 1, [134].log_data[1].valid := 1, [134].log_data[2].valid := 1, [134].log_data[3].valid := 1, [134].log_data[4].valid := 1, [134].log_data[5].valid := 1, [134].log_data[6].valid := 1, [134].log_data[7].valid := 1, [134].log_data[8].valid := 1, [134].log_data[9].valid := 1, [134].log_data[10].valid := 1, [134].log_data[11].valid := 1, [134].log_data[12].valid := 1, [134].log_data[13].valid := 1, [134].log_data[14].valid := 1, [134].log_data[15].valid := 1, [134].log_data[16].valid := 1, [134].log_data[17].valid := 1, [134].log_data[18].valid := 1, [134].log_data[19].valid := 1, [134].time.Year := 2023, [134].time.Month := 1, [134].time.Day := 18, [134].time.Hour := 11, [134].time.Minute := 34, [134].time.Second := 59, [135].log_data[0].min := 1.0, [135].log_data[0].max := 1.0, [135].log_data[0].total := 300.0, [135].log_data[0].time := 300.0, [135].log_data[0].minminute := 35, [135].log_data[0].maxminute := 35, [135].log_data[0].valid := 1, [135].log_data[1].valid := 1, [135].log_data[2].valid := 1, [135].log_data[3].valid := 1, [135].log_data[4].valid := 1, [135].log_data[5].valid := 1, [135].log_data[6].valid := 1, [135].log_data[7].valid := 1, [135].log_data[8].valid := 1, [135].log_data[9].valid := 1, [135].log_data[10].valid := 1, [135].log_data[11].valid := 1, [135].log_data[12].valid := 1, [135].log_data[13].valid := 1, [135].log_data[14].valid := 1, [135].log_data[15].valid := 1, [135].log_data[16].valid := 1, [135].log_data[17].valid := 1, [135].log_data[18].valid := 1, [135].log_data[19].valid := 1, [135].time.Year := 2023, [135].time.Month := 1, [135].time.Day := 18, [135].time.Hour := 11,
        [135].time.Minute := 39, [135].time.Second := 59, [136].log_data[0].min := 1.0, [136].log_data[0].max := 1.0, [136].log_data[0].total := 300.0, [136].log_data[0].time := 300.0, [136].log_data[0].minminute := 40, [136].log_data[0].maxminute := 40, [136].log_data[0].valid := 1, [136].log_data[1].valid := 1, [136].log_data[2].valid := 1, [136].log_data[3].valid := 1, [136].log_data[4].valid := 1, [136].log_data[5].valid := 1, [136].log_data[6].valid := 1, [136].log_data[7].valid := 1, [136].log_data[8].valid := 1, [136].log_data[9].valid := 1, [136].log_data[10].valid := 1, [136].log_data[11].valid := 1, [136].log_data[12].valid := 1, [136].log_data[13].valid := 1, [136].log_data[14].valid := 1, [136].log_data[15].valid := 1, [136].log_data[16].valid := 1, [136].log_data[17].valid := 1, [136].log_data[18].valid := 1, [136].log_data[19].valid := 1, [136].time.Year := 2023, [136].time.Month := 1, [136].time.Day := 18, [136].time.Hour := 11, [136].time.Minute := 44, [136].time.Second := 59, [137].log_data[0].min := 1.0, [137].log_data[0].max := 1.0, [137].log_data[0].total := 300.0, [137].log_data[0].time := 300.0, [137].log_data[0].minminute := 45, [137].log_data[0].maxminute := 45, [137].log_data[0].valid := 1, [137].log_data[1].valid := 1, [137].log_data[2].valid := 1, [137].log_data[3].valid := 1, [137].log_data[4].valid := 1, [137].log_data[5].valid := 1, [137].log_data[6].valid := 1, [137].log_data[7].valid := 1, [137].log_data[8].valid := 1, [137].log_data[9].valid := 1, [137].log_data[10].valid := 1, [137].log_data[11].valid := 1, [137].log_data[12].valid := 1, [137].log_data[13].valid := 1, [137].log_data[14].valid := 1, [137].log_data[15].valid := 1, [137].log_data[16].valid := 1, [137].log_data[17].valid := 1, [137].log_data[18].valid := 1, [137].log_data[19].valid := 1,
        [137].time.Year := 2023, [137].time.Month := 1, [137].time.Day := 18, [137].time.Hour := 11, [137].time.Minute := 49, [137].time.Second := 59, [138].log_data[0].min := 1.0, [138].log_data[0].max := 1.0, [138].log_data[0].total := 300.0, [138].log_data[0].time := 300.0, [138].log_data[0].minminute := 50, [138].log_data[0].maxminute := 50, [138].log_data[0].valid := 1, [138].log_data[1].valid := 1, [138].log_data[2].valid := 1, [138].log_data[3].valid := 1, [138].log_data[4].valid := 1, [138].log_data[5].valid := 1, [138].log_data[6].valid := 1, [138].log_data[7].valid := 1, [138].log_data[8].valid := 1, [138].log_data[9].valid := 1, [138].log_data[10].valid := 1, [138].log_data[11].valid := 1, [138].log_data[12].valid := 1, [138].log_data[13].valid := 1, [138].log_data[14].valid := 1, [138].log_data[15].valid := 1, [138].log_data[16].valid := 1, [138].log_data[17].valid := 1, [138].log_data[18].valid := 1, [138].log_data[19].valid := 1, [138].time.Year := 2023, [138].time.Month := 1, [138].time.Day := 18, [138].time.Hour := 11, [138].time.Minute := 54, [138].time.Second := 59, [139].log_data[0].min := 1.0, [139].log_data[0].max := 1.0, [139].log_data[0].total := 300.0, [139].log_data[0].time := 300.0, [139].log_data[0].minminute := 55, [139].log_data[0].maxminute := 55, [139].log_data[0].valid := 1, [139].log_data[1].valid := 1, [139].log_data[2].valid := 1, [139].log_data[3].valid := 1, [139].log_data[4].valid := 1, [139].log_data[5].valid := 1, [139].log_data[6].valid := 1, [139].log_data[7].valid := 1, [139].log_data[8].valid := 1, [139].log_data[9].valid := 1, [139].log_data[10].valid := 1, [139].log_data[11].valid := 1, [139].log_data[12].valid := 1, [139].log_data[13].valid := 1, [139].log_data[14].valid := 1, [139].log_data[15].valid := 1,
        [139].log_data[16].valid := 1, [139].log_data[17].valid := 1, [139].log_data[18].valid := 1, [139].log_data[19].valid := 1, [139].time.Year := 2023, [139].time.Month := 1, [139].time.Day := 18, [139].time.Hour := 11, [139].time.Minute := 59, [139].time.Second := 59, [140].log_data[0].min := 1.0, [140].log_data[0].max := 1.0, [140].log_data[0].total := 300.0, [140].log_data[0].time := 300.0, [140].log_data[0].valid := 1, [140].log_data[1].valid := 1, [140].log_data[2].valid := 1, [140].log_data[3].valid := 1, [140].log_data[4].valid := 1, [140].log_data[5].valid := 1, [140].log_data[6].valid := 1, [140].log_data[7].valid := 1, [140].log_data[8].valid := 1, [140].log_data[9].valid := 1, [140].log_data[10].valid := 1, [140].log_data[11].valid := 1, [140].log_data[12].valid := 1, [140].log_data[13].valid := 1, [140].log_data[14].valid := 1, [140].log_data[15].valid := 1, [140].log_data[16].valid := 1, [140].log_data[17].valid := 1, [140].log_data[18].valid := 1, [140].log_data[19].valid := 1, [140].time.Year := 2023, [140].time.Month := 1, [140].time.Day := 18, [140].time.Hour := 12, [140].time.Minute := 4, [140].time.Second := 59, [141].log_data[0].min := 1.0, [141].log_data[0].max := 1.0, [141].log_data[0].total := 300.0, [141].log_data[0].time := 300.0, [141].log_data[0].minminute := 5, [141].log_data[0].maxminute := 5, [141].log_data[0].valid := 1, [141].log_data[1].valid := 1, [141].log_data[2].valid := 1, [141].log_data[3].valid := 1, [141].log_data[4].valid := 1, [141].log_data[5].valid := 1, [141].log_data[6].valid := 1, [141].log_data[7].valid := 1, [141].log_data[8].valid := 1, [141].log_data[9].valid := 1, [141].log_data[10].valid := 1, [141].log_data[11].valid := 1, [141].log_data[12].valid := 1, [141].log_data[13].valid := 1,
        [141].log_data[14].valid := 1, [141].log_data[15].valid := 1, [141].log_data[16].valid := 1, [141].log_data[17].valid := 1, [141].log_data[18].valid := 1, [141].log_data[19].valid := 1, [141].time.Year := 2023, [141].time.Month := 1, [141].time.Day := 18, [141].time.Hour := 12, [141].time.Minute := 9, [141].time.Second := 59, [142].log_data[0].min := 1.0, [142].log_data[0].max := 1.0, [142].log_data[0].total := 300.0, [142].log_data[0].time := 300.0, [142].log_data[0].minminute := 10, [142].log_data[0].maxminute := 10, [142].log_data[0].valid := 1, [142].log_data[1].valid := 1, [142].log_data[2].valid := 1, [142].log_data[3].valid := 1, [142].log_data[4].valid := 1, [142].log_data[5].valid := 1, [142].log_data[6].valid := 1, [142].log_data[7].valid := 1, [142].log_data[8].valid := 1, [142].log_data[9].valid := 1, [142].log_data[10].valid := 1, [142].log_data[11].valid := 1, [142].log_data[12].valid := 1, [142].log_data[13].valid := 1, [142].log_data[14].valid := 1, [142].log_data[15].valid := 1, [142].log_data[16].valid := 1, [142].log_data[17].valid := 1, [142].log_data[18].valid := 1, [142].log_data[19].valid := 1, [142].time.Year := 2023, [142].time.Month := 1, [142].time.Day := 18, [142].time.Hour := 12, [142].time.Minute := 14, [142].time.Second := 59, [143].log_data[0].min := 1.0, [143].log_data[0].max := 1.0, [143].log_data[0].total := 300.0, [143].log_data[0].time := 300.0, [143].log_data[0].minminute := 15, [143].log_data[0].maxminute := 15, [143].log_data[0].valid := 1, [143].log_data[1].valid := 1, [143].log_data[2].valid := 1, [143].log_data[3].valid := 1, [143].log_data[4].valid := 1, [143].log_data[5].valid := 1, [143].log_data[6].valid := 1, [143].log_data[7].valid := 1, [143].log_data[8].valid := 1, [143].log_data[9].valid := 1,
        [143].log_data[10].valid := 1, [143].log_data[11].valid := 1, [143].log_data[12].valid := 1, [143].log_data[13].valid := 1, [143].log_data[14].valid := 1, [143].log_data[15].valid := 1, [143].log_data[16].valid := 1, [143].log_data[17].valid := 1, [143].log_data[18].valid := 1, [143].log_data[19].valid := 1, [143].time.Year := 2023, [143].time.Month := 1, [143].time.Day := 18, [143].time.Hour := 12, [143].time.Minute := 19, [143].time.Second := 59, [144].log_data[0].min := 1.0, [144].log_data[0].max := 1.0, [144].log_data[0].total := 300.0, [144].log_data[0].time := 300.0, [144].log_data[0].minminute := 20, [144].log_data[0].maxminute := 20, [144].log_data[0].valid := 1, [144].log_data[1].valid := 1, [144].log_data[2].valid := 1, [144].log_data[3].valid := 1, [144].log_data[4].valid := 1, [144].log_data[5].valid := 1, [144].log_data[6].valid := 1, [144].log_data[7].valid := 1, [144].log_data[8].valid := 1, [144].log_data[9].valid := 1, [144].log_data[10].valid := 1, [144].log_data[11].valid := 1, [144].log_data[12].valid := 1, [144].log_data[13].valid := 1, [144].log_data[14].valid := 1, [144].log_data[15].valid := 1, [144].log_data[16].valid := 1, [144].log_data[17].valid := 1, [144].log_data[18].valid := 1, [144].log_data[19].valid := 1, [144].time.Year := 2023, [144].time.Month := 1, [144].time.Day := 18, [144].time.Hour := 12, [144].time.Minute := 24, [144].time.Second := 59, [145].log_data[0].min := 1.0, [145].log_data[0].max := 1.0, [145].log_data[0].total := 300.0, [145].log_data[0].time := 300.0, [145].log_data[0].minminute := 25, [145].log_data[0].maxminute := 25, [145].log_data[0].valid := 1, [145].log_data[1].valid := 1, [145].log_data[2].valid := 1, [145].log_data[3].valid := 1, [145].log_data[4].valid := 1, [145].log_data[5].valid := 1,
        [145].log_data[6].valid := 1, [145].log_data[7].valid := 1, [145].log_data[8].valid := 1, [145].log_data[9].valid := 1, [145].log_data[10].valid := 1, [145].log_data[11].valid := 1, [145].log_data[12].valid := 1, [145].log_data[13].valid := 1, [145].log_data[14].valid := 1, [145].log_data[15].valid := 1, [145].log_data[16].valid := 1, [145].log_data[17].valid := 1, [145].log_data[18].valid := 1, [145].log_data[19].valid := 1, [145].time.Year := 2023, [145].time.Month := 1, [145].time.Day := 18, [145].time.Hour := 12, [145].time.Minute := 29, [145].time.Second := 59, [146].log_data[0].min := 1.0, [146].log_data[0].max := 1.0, [146].log_data[0].total := 300.0, [146].log_data[0].time := 300.0, [146].log_data[0].minminute := 30, [146].log_data[0].maxminute := 30, [146].log_data[0].valid := 1, [146].log_data[1].valid := 1, [146].log_data[2].valid := 1, [146].log_data[3].valid := 1, [146].log_data[4].valid := 1, [146].log_data[5].valid := 1, [146].log_data[6].valid := 1, [146].log_data[7].valid := 1, [146].log_data[8].valid := 1, [146].log_data[9].valid := 1, [146].log_data[10].valid := 1, [146].log_data[11].valid := 1, [146].log_data[12].valid := 1, [146].log_data[13].valid := 1, [146].log_data[14].valid := 1, [146].log_data[15].valid := 1, [146].log_data[16].valid := 1, [146].log_data[17].valid := 1, [146].log_data[18].valid := 1, [146].log_data[19].valid := 1, [146].time.Year := 2023, [146].time.Month := 1, [146].time.Day := 18, [146].time.Hour := 12, [146].time.Minute := 34, [146].time.Second := 59, [147].log_data[0].min := 1.0, [147].log_data[0].max := 1.0, [147].log_data[0].total := 300.0, [147].log_data[0].time := 300.0, [147].log_data[0].minminute := 35, [147].log_data[0].maxminute := 35, [147].log_data[0].valid := 1, [147].log_data[1].valid := 1,
        [147].log_data[2].valid := 1, [147].log_data[3].valid := 1, [147].log_data[4].valid := 1, [147].log_data[5].valid := 1, [147].log_data[6].valid := 1, [147].log_data[7].valid := 1, [147].log_data[8].valid := 1, [147].log_data[9].valid := 1, [147].log_data[10].valid := 1, [147].log_data[11].valid := 1, [147].log_data[12].valid := 1, [147].log_data[13].valid := 1, [147].log_data[14].valid := 1, [147].log_data[15].valid := 1, [147].log_data[16].valid := 1, [147].log_data[17].valid := 1, [147].log_data[18].valid := 1, [147].log_data[19].valid := 1, [147].time.Year := 2023, [147].time.Month := 1, [147].time.Day := 18, [147].time.Hour := 12, [147].time.Minute := 39, [147].time.Second := 59, [148].log_data[0].min := 1.0, [148].log_data[0].max := 1.0, [148].log_data[0].total := 300.0, [148].log_data[0].time := 300.0, [148].log_data[0].minminute := 40, [148].log_data[0].maxminute := 40, [148].log_data[0].valid := 1, [148].log_data[1].valid := 1, [148].log_data[2].valid := 1, [148].log_data[3].valid := 1, [148].log_data[4].valid := 1, [148].log_data[5].valid := 1, [148].log_data[6].valid := 1, [148].log_data[7].valid := 1, [148].log_data[8].valid := 1, [148].log_data[9].valid := 1, [148].log_data[10].valid := 1, [148].log_data[11].valid := 1, [148].log_data[12].valid := 1, [148].log_data[13].valid := 1, [148].log_data[14].valid := 1, [148].log_data[15].valid := 1, [148].log_data[16].valid := 1, [148].log_data[17].valid := 1, [148].log_data[18].valid := 1, [148].log_data[19].valid := 1, [148].time.Year := 2023, [148].time.Month := 1, [148].time.Day := 18, [148].time.Hour := 12, [148].time.Minute := 44, [148].time.Second := 59, [149].log_data[0].min := 1.0, [149].log_data[0].max := 1.0, [149].log_data[0].total := 300.0, [149].log_data[0].time := 300.0,
